(* CODESYS project Rasi_feeds_batching2.project

Project tree, tasks and I/O mapping:
  PLC_AC500_V3 : PM5032-T-ETH, ABB AG, order no. 1SAP123400R0x72, version 3.7.0.0
    application Application
      libraries: ModbusRtu, * (ABB); Util, * (System)
      task Task (cyclic, interval t#10ms, priority 14, watchdog t#20ms x 1) calls batching14
      CheckConfigurationObject
      Diagnosis/
        text list Diag_IO_Bus
        text list Diag_V3_PLC
      global variables GVL
      function block Auto_Batching_V14 [ST]
      function block Semi_Auto_Batching_V14 [ST]
      function block FB_Samyak_Multi [ST]
      function block FB_Samyak_Control [ST]
      function block Auto_Batching_V15 [ST]
      function block Semi_Auto_Batching_V15 [ST]
      program batching14 [FBD]
    OnBoard_IO : 12DI/8DO-T/2DC, ABB AG, version 3.7.0.0
        input  E_Stop_DI : BOOL  // Fast inputs DI0-DI3.Digital input DI0
        input  Main_Cont_FB : BOOL  // Fast inputs DI0-DI3.Digital input DI1
        input  Auto_Mode_FB : BOOL  // Fast inputs DI0-DI3.Digital input DI2
        input  VFD_Run : BOOL  // Fast inputs DI0-DI3.Digital input DI3
        input  Start_PB : BOOL  // Fast inputs DI4-DI7.Digital input DI4
        unmapped channels: Fast inputs DI0-DI3, Fast inputs DI4-DI7, Standard inputs DI8-DI11, Digital inputs - Transistor, Fast outputs DO0-DO3, Fast outputs DO4-DO7, Digital outputs - Transistor
    IO_Bus : I/O-Bus, ABB AG, version 3.7.0.0
    Interfaces : Interfaces, ABB AG, version 3.7.0.0
      TA5142_RS485I : TA5142-RS485I, ABB AG, order no. 1SAP187300R0x02, version 3.7.0.0
        Modbus_RTU_Client : Modbus RTU Client, ABB AG, version 3.7.0.0
      OptionSlot_2
      Ethernet : Ethernet, ABB AG, version 3.7.0.0
        ETH1 : IP Settings, ABB AG, version 3.7.0.0
          NetConfig : NetConfig, ABB AG, version 3.7.0.0
          Modbus_TCP_IP_Server : Modbus TCP/IP Server, ABB AG, version 3.7.0.0
        Protocols : Client Protocols, ABB AG, version 3.7.0.0
    OnBoard_RTC : OnBoard RTC, ABB AG, version 3.7.0.0
  text list GlobalTextList
*)

// PLC_AC500_V3/Application/GVL
{attribute 'qualified_only'}
VAR_GLOBAL
    Recipe_Weights AT %MD100 : ARRAY[1..20] OF REAL;
	Auto_Bin_Material_Mapping AT %MW50: ARRAY[1..6] OF INT;
	Semi_Auto_Bin_Material_Mapping AT %MW60: ARRAY[1..10] OF INT;
	Auto_Coarse_To_Fine_speed AT %MD120: ARRAY[1..6] OF REAL := [1.0,1.0,1.0,1.0,1.0,1.0];
	Semi_Auto_Coarse_To_Fine_speed AT %MD130: ARRAY[1..10] OF REAL := [1.0,1.0,1.0,1.0,1.0,1.0,1.0,1.0,1.0,1.0];
	Auto_Bin_Tolerance AT %MD150: ARRAY[1..6] OF REAL;
	Semi_Auto_Bin_Tolerance AT %MD160: ARRAY[1..10] OF REAL;
	Start_Button AT %MX2.0: BOOL;
	E_Stop_Active AT %MX2.1: BOOL;
	Reset AT %MX2.3: BOOL;
	Next_Cycle_Start AT %MX2.4: BOOL;               // Command pulse/signal to start next batch cycle after hoppers are emptied
	Auto_Active_Mat AT %MW70: INT;
	Auto_Active_Bin AT %MW71: INT;
	Semi_Auto_Active_Mat AT %MW72: INT;
	Semi_Auto_Active_Bin AT %MW73: INT;
	Target_Batch_Cycles AT %MW74: INT := 1;
	Current_Batch_Cycle AT %MW75: INT;
	Completed_Batch_Cycles AT %MW79: INT;
	Error_Code AT %MW76: INT;  // 0=OK 1=DupMat 2=MatRange 3=RecipeLimit 4=ScaleNotEmpty 5=CommunicationFault(Line_Fault) 6=Ex_Weight_Allow_kg_invalid 21=ScaleOverload
	Run AT %MX2.5 : BOOL;
	load_cell_auto AT %MD174 : REAL;
	load_cell_semi_auto AT %MD175 : REAL;
	Auto_Initial_Tolerance AT %MD176 : REAL := 5.0;
	Semi_Auto_Initial_Tolerance AT %MD178 : REAL := 5.0;
	Empty_Weight_Limit AT %MD186 : REAL := 5.0;     // Maximum scale weight limit (kg) to qualify scale as empty before starting next cycle
	Ex_Weight_Allow_kg AT %MD188 : REAL := 0.2;  // Semi-only: oscillation allow (kg) above target; next stage only if actual < Target+Allow
	Auto_Total_Target_Weight AT %MD170 : REAL;
	Semi_Auto_Total_Target_Weight AT %MD171 : REAL;
	Auto_Material_Count AT %MW77: INT;
	Semi_Auto_Material_Count AT %MW78 : INT;
	Auto_Current_Step AT %MW80 : INT;
	Semi_Auto_Current_Step AT %MW81 : INT;
	Auto_Active_Target_Weight AT %MD220 : REAL;
	Semi_Auto_Active_Target_Weight AT %MD224 : REAL;
	Auto_Active_Live_Weight AT %MD172 : REAL;
	Semi_Auto_Active_Live_Weight AT %MD173 : REAL;
	Auto_Excess_Allowed AT %MX2.6: BOOL := 1;
	Semi_Auto_Excess_Allowed AT %MX2.9 : BOOL;
	Auto_Excess_Alarm AT %MX2.7 : BOOL;
	Semi_Auto_Excess_Alarm AT %MX2.8 : BOOL;
	Auto_Inter_Bin_Delay AT %MD190 : TIME;
	Semi_Auto_Inter_Bin_Delay AT %MD194 : TIME;
	Auto_Sequence_Complete AT %MX3.0 : BOOL;
	Semi_Auto_Sequence_Complete AT %MX3.1 : BOOL;
	All_Cycles_Complete AT %MX3.2 : BOOL;           // Master flag: TRUE when all target batch cycles have completed
	Auto_Status_Message : STRING(80);
	Semi_Auto_Status_Message : STRING(80);
	
	(* 8 Process Output and Weight Arrays *)
	Auto_Bin : ARRAY[1..6] OF BOOL;
	auto_bin_cutoff : ARRAY[1..6] OF BOOL;
	auto_bin_motor : ARRAY[1..6] OF BOOL;
	Semi_Auto_Bin : ARRAY[1..10] OF BOOL;
	semi_auto_bin_cutoff : ARRAY[1..10] OF BOOL;
	semi_auto_bin_motor : ARRAY[1..10] OF BOOL;
	Auto_Weights : ARRAY[1..6] OF REAL;
	Semi_Auto_Weights : ARRAY[1..10] OF REAL;
	Waiting_Next_batch_HMI_HIDE AT %MX8.1: BOOL;
END_VAR

// PLC_AC500_V3/Application/batching14
PROGRAM batching14
VAR
	Auto_Ctrl: Auto_Batching_V15;
	Semi_Auto_Ctrl: Semi_Auto_Batching_V15;
	Auto_Complete: BOOL;
	Semi_Auto_Complete: BOOL;
	Auto_Err: INT;
	Auto_Msg: STRING;
	Semi_Auto_Err: INT;
	Semi_Auto_Msg: STRING;
	AutoBatchScale: MODRTUMAST;
	ModEnabler: BLINK;
	SamyakRaw: ARRAY[0..1] OF DINT;
	AutBatchRaw: ARRAY[0..1] OF DINT;
	SemAutoScale: MODRTUMAST;
	SemiAutoScaleRaw: ARRAY[0..1] OF DINT;
	AutoBatchSamyak: REAL;
	FB_Samyak_Multi_1: FB_Samyak_Multi;
	FB_Samyak_Control_1: FB_Samyak_Control;
	Run_PB_1: BOOL;
	Next_Cycle_Start: BOOL;
	TP_1: TP;
	TP_ON: BOOL;
	TP_Out: BOOL;
	TP_Et: TIME;
	arrTare_Cmds: ARRAY[1..4] OF BOOL;
END_VAR

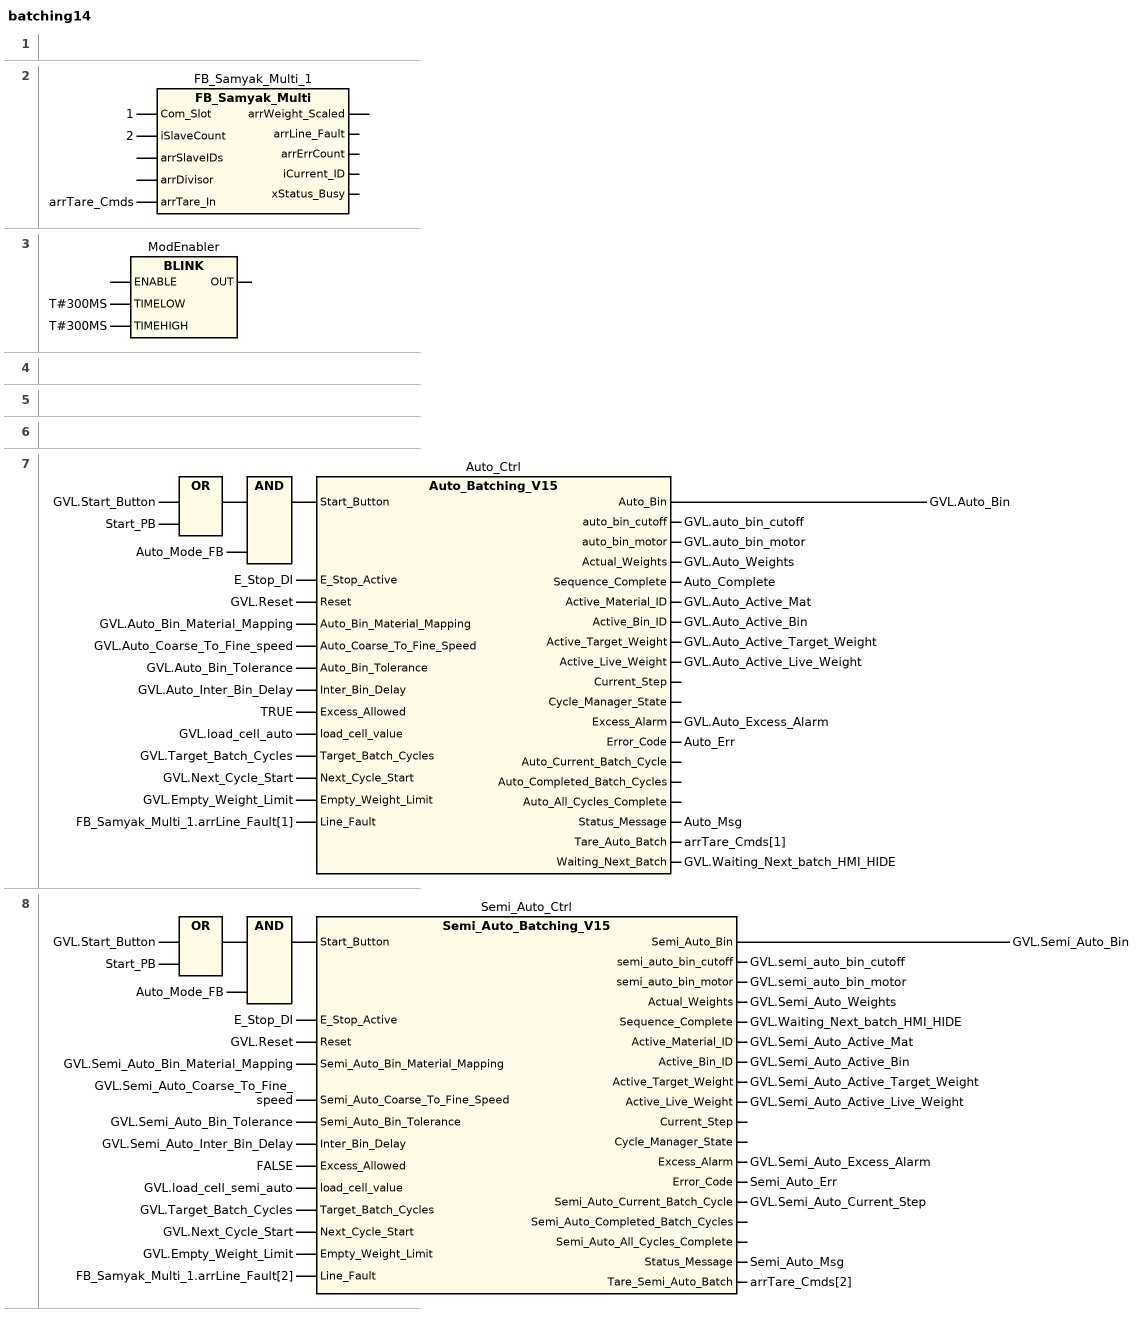
// NETWORK 1

// NETWORK 2
FB_Samyak_Multi_1(Com_Slot := 1, iSlaveCount := 2, arrTare_In := arrTare_Cmds); // FB_Samyak_Multi

// NETWORK 3
ModEnabler(TIMELOW := T#300MS, TIMEHIGH := T#300MS); // BLINK

// NETWORK 4

// NETWORK 5

// NETWORK 6

// NETWORK 7
Auto_Ctrl(
    Start_Button := (GVL.Start_Button OR Start_PB) AND Auto_Mode_FB,
    E_Stop_Active := E_Stop_DI,
    Reset := GVL.Reset,
    Auto_Bin_Material_Mapping := GVL.Auto_Bin_Material_Mapping,
    Auto_Coarse_To_Fine_Speed := GVL.Auto_Coarse_To_Fine_speed,
    Auto_Bin_Tolerance := GVL.Auto_Bin_Tolerance,
    Inter_Bin_Delay := GVL.Auto_Inter_Bin_Delay,
    Excess_Allowed := TRUE,
    load_cell_value := GVL.load_cell_auto,
    Target_Batch_Cycles := GVL.Target_Batch_Cycles,
    Next_Cycle_Start := GVL.Next_Cycle_Start,
    Empty_Weight_Limit := GVL.Empty_Weight_Limit,
    Line_Fault := FB_Samyak_Multi_1.arrLine_Fault[1],
    auto_bin_cutoff => GVL.auto_bin_cutoff,
    auto_bin_motor => GVL.auto_bin_motor,
    Actual_Weights => GVL.Auto_Weights,
    Sequence_Complete => Auto_Complete,
    Active_Material_ID => GVL.Auto_Active_Mat,
    Active_Bin_ID => GVL.Auto_Active_Bin,
    Active_Target_Weight => GVL.Auto_Active_Target_Weight,
    Active_Live_Weight => GVL.Auto_Active_Live_Weight,
    Excess_Alarm => GVL.Auto_Excess_Alarm,
    Error_Code => Auto_Err,
    Status_Message => Auto_Msg,
    Tare_Auto_Batch => arrTare_Cmds[1],
    Waiting_Next_Batch => GVL.Waiting_Next_batch_HMI_HIDE); // Auto_Batching_V15
GVL.Auto_Bin := Auto_Ctrl.Auto_Bin;

// NETWORK 8
Semi_Auto_Ctrl(
    Start_Button := (GVL.Start_Button OR Start_PB) AND Auto_Mode_FB,
    E_Stop_Active := E_Stop_DI,
    Reset := GVL.Reset,
    Semi_Auto_Bin_Material_Mapping := GVL.Semi_Auto_Bin_Material_Mapping,
    Semi_Auto_Coarse_To_Fine_Speed := GVL.Semi_Auto_Coarse_To_Fine_speed,
    Semi_Auto_Bin_Tolerance := GVL.Semi_Auto_Bin_Tolerance,
    Inter_Bin_Delay := GVL.Semi_Auto_Inter_Bin_Delay,
    Excess_Allowed := FALSE,
    load_cell_value := GVL.load_cell_semi_auto,
    Target_Batch_Cycles := GVL.Target_Batch_Cycles,
    Next_Cycle_Start := GVL.Next_Cycle_Start,
    Empty_Weight_Limit := GVL.Empty_Weight_Limit,
    Line_Fault := FB_Samyak_Multi_1.arrLine_Fault[2],
    semi_auto_bin_cutoff => GVL.semi_auto_bin_cutoff,
    semi_auto_bin_motor => GVL.semi_auto_bin_motor,
    Actual_Weights => GVL.Semi_Auto_Weights,
    Sequence_Complete => GVL.Waiting_Next_batch_HMI_HIDE,
    Active_Material_ID => GVL.Semi_Auto_Active_Mat,
    Active_Bin_ID => GVL.Semi_Auto_Active_Bin,
    Active_Target_Weight => GVL.Semi_Auto_Active_Target_Weight,
    Active_Live_Weight => GVL.Semi_Auto_Active_Live_Weight,
    Excess_Alarm => GVL.Semi_Auto_Excess_Alarm,
    Error_Code => Semi_Auto_Err,
    Semi_Auto_Current_Batch_Cycle => GVL.Semi_Auto_Current_Step,
    Status_Message => Semi_Auto_Msg,
    Tare_Semi_Auto_Batch => arrTare_Cmds[2]); // Semi_Auto_Batching_V15
GVL.Semi_Auto_Bin := Semi_Auto_Ctrl.Semi_Auto_Bin;

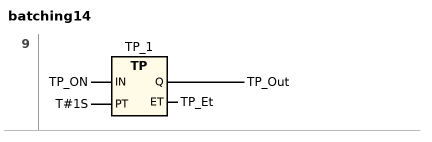
// NETWORK 9
TP_1(IN := TP_ON, PT := T#1S, ET => TP_Et); // TP
TP_Out := TP_1.Q;

END_PROGRAM

// PLC_AC500_V3/Application/FB_Samyak_Multi
//SAMYAK 4016 Multi Slave Unit Customised Block
//Note: This FB_Samyak_Multi name is impotrtant when you create new POU.

FUNCTION_BLOCK FB_Samyak_Multi
VAR_INPUT
    Com_Slot      : BYTE := 1;    (* Port Number *)
    iSlaveCount   : INT := 1;     (* How many slaves active: 1 to 4 *)
    arrSlaveIDs   : ARRAY[1..4] OF BYTE := [1, 2, 3, 4]; (* Unit IDs *)
    arrDivisor    : ARRAY[1..4] OF REAL := [10.0, 10.0, 10.0, 10.0]; (* Scaling per Unit *)
    arrTare_In    : ARRAY[1..4] OF BOOL; (* Individual Tare triggers *)
END_VAR

VAR_OUTPUT
    arrWeight_Scaled : ARRAY[1..4] OF REAL; (* Scaled result per unit *)
    arrLine_Fault    : ARRAY[1..4] OF BOOL; (* Fault status per unit *)
    arrErrCount      : ARRAY[1..4] OF INT;  (* Error count per unit *)
    iCurrent_ID      : BYTE;                (* Current ID being polled *)
    xStatus_Busy     : BOOL;                (* Overall Bus Busy *)
END_VAR

VAR
    (* Internal ModRtuMast Instances *)
    fbRead         : ModRtuMast;
    fbTare         : ModRtuMast;
    
    (* Polling Control *)
    iStep          : INT := 0;
    iIdx           : INT := 1;    (* Current Loop Index *)
    Samyak_Buffer  : ARRAY[0..17] OF WORD;
    wTareCommand   : WORD := 1;
    
    (* Unique Timer/Trigger Instances *)
    rtTareTrig     : R_TRIG;
    rtErrTrig      : R_TRIG;
    tWatchdog      : TON;
    tRecovery      : TON;
END_VAR



(* --- 1. INDIVIDUAL UNIT MONITORING --- *)
iCurrent_ID := arrSlaveIDs[iIdx]; 

(* Watchdog for Bus Hangs *)
tWatchdog(IN := (fbRead.Busy OR fbTare.Busy), PT := T#2000MS);
xStatus_Busy := fbRead.Busy OR fbTare.Busy;

(* Error Tracking for Current Index *)
rtErrTrig(CLK := (fbRead.Error OR fbTare.Error));
IF rtErrTrig.Q THEN
    arrErrCount[iIdx] := arrErrCount[iIdx] + 1;
END_IF

(* Reset on Success *)
IF fbRead.Done OR fbTare.Done THEN
    arrErrCount[iIdx] := 0;
    arrLine_Fault[iIdx] := FALSE;
END_IF

(* Line Fault Activation (10 errors) *)
IF arrErrCount[iIdx] >= 10 THEN
    arrLine_Fault[iIdx] := TRUE;
END_IF

(* Auto-Recovery pulse (5s) *)
tRecovery(IN := arrLine_Fault[iIdx], PT := T#5S);
IF tRecovery.Q THEN
    arrErrCount[iIdx] := 0;
    arrLine_Fault[iIdx] := FALSE;
END_IF

IF tWatchdog.Q THEN iStep := 99; END_IF

(* Check Tare for active slave *)
rtTareTrig(CLK := arrTare_In[iIdx]);

(* --- 2. SEQUENTIAL STATE MACHINE --- *)
CASE iStep OF
    
    0: (* READ CURRENT SLAVE *)
        fbTare(Execute := FALSE);
        fbRead(
            Execute := NOT (fbRead.Done OR fbRead.Error OR fbRead.Busy) 
                       AND NOT rtTareTrig.Q AND NOT arrLine_Fault[iIdx],
            COM     := Com_Slot,
            Serv    := arrSlaveIDs[iIdx],
            FCT     := 3, Addr := 0, Nb := 2, 
            Data    := ADR(Samyak_Buffer[0]), Timeout := 400
        );

        IF fbRead.Done THEN
            (* Scale weight using the array-based divisor for this specific index *)
            arrWeight_Scaled[iIdx] := TO_REAL(TO_DINT(SHL(TO_DWORD(Samyak_Buffer[1]), 16) OR TO_DWORD(Samyak_Buffer[0]))) / arrDivisor[iIdx];
            iStep := 10; (* Switch to next slave *)
        END_IF
        
        IF fbRead.Error THEN iStep := 10; END_IF (* Move on if error *)
        IF rtTareTrig.Q THEN iStep := 1; END_IF  (* Priority: Tare current unit *)

    1: (* PORT RELEASE *)
        fbRead(Execute := FALSE);
        IF NOT fbRead.Busy THEN iStep := 2; END_IF

    2: (* WRITE TARE FOR CURRENT SLAVE *)
        fbTare(
            Execute := TRUE,
            COM := Com_Slot, Serv := arrSlaveIDs[iIdx], 
            FCT := 6, Addr := 16, Nb := 1,
            Data := ADR(wTareCommand), Timeout := 1000
        );

        IF fbTare.Done OR fbTare.Error THEN
            arrTare_In[iIdx] := FALSE; (* Reset manual trigger *)
            iStep := 3;
        END_IF

    3: (* CLEANUP *)
        fbTare(Execute := FALSE);
        IF NOT fbTare.Busy THEN iStep := 10; END_IF

    10: (* INDEX ROTATION *)
        iIdx := iIdx + 1;
        IF iIdx > iSlaveCount THEN
            iIdx := 1; (* Back to first slave *)
        END_IF
        iStep := 0;

    99: (* EMERGENCY RESET *)
        fbRead(Execute := FALSE); fbTare(Execute := FALSE);
        IF NOT (fbRead.Busy OR fbTare.Busy) THEN iStep := 0; END_IF
        
END_CASE

END_FUNCTION_BLOCK

// PLC_AC500_V3/Application/Auto_Batching_V15
FUNCTION_BLOCK Auto_Batching_V15
VAR_INPUT
    Start_Button : BOOL;                            // Command pulse/signal to start or resume the auto batching sequence
    E_Stop_Active : BOOL;                           // Emergency Stop circuit status (NC contact: TRUE = Healthy/Run permitted, FALSE = E-Stop tripped)
    Reset : BOOL;                                   // System reset pulse (clears active steps, outputs, alarms, and error flags)
    Auto_Bin_Material_Mapping : ARRAY[1..6] OF INT; // Array mapping physical Silos 1..6 to Recipe Material IDs (1..20, 0 = Silo skipped)
    Auto_Coarse_To_Fine_Speed : ARRAY[1..6] OF REAL;// Weight offset threshold (kg) before target to transition from Coarse to Fine feeding
    Auto_Bin_Tolerance : ARRAY[1..6] OF REAL;       // Allowable weight tolerance window (±kg) around target weight for each silo
    Inter_Bin_Delay : TIME;                         // Settling delay duration after completing a bin before advancing to the next
    Excess_Allowed : BOOL;                          // Overfill handling policy: TRUE = proceed if target is exceeded, FALSE = raise alarm and halt
    load_cell_value : REAL;                         // Live gross weight input reading from the Auto scale load cell (kg)
    Target_Batch_Cycles : INT;                      // Target number of batch cycle repetitions configured from HMI (defaults to 1)
    Next_Cycle_Start : BOOL;                        // NextBatchStart: after a completed cycle (Target>1), press when this FB scale < Empty_Weight_Limit
    Empty_Weight_Limit : REAL;                      // Tank minimum / empty limit (kg): load_cell must be LT this before Next_Cycle_Start is accepted
    Line_Fault : BOOL;                              // Wire from FB_Samyak_Multi.arrLine_Fault[n] (Auto scale). TRUE = hold process (Over Dump Avoid)
END_VAR
VAR_OUTPUT
    Auto_Bin : ARRAY[1..6] OF BOOL;                 // Coarse feeding valve / gate actuation command outputs for Silos 1..6
    auto_bin_cutoff : ARRAY[1..6] OF BOOL;          // Fine feeding valve / vibrator cutoff actuation command outputs for Silos 1..6
    auto_bin_motor : ARRAY[1..6] OF BOOL;           // Feeder / screw conveyor motor run commands for Silos 1..6
    Actual_Weights : ARRAY[1..6] OF REAL;           // Net material weight (kg) successfully dosed for each silo in the current cycle
    Sequence_Complete : BOOL;                       // Handshake flag: TRUE when all mapped Auto silos have completed dosing and settling
    Active_Material_ID : INT;                       // Recipe Material ID currently being dosed (1..20, 0 when idle/complete)
    Active_Bin_ID : INT;                            // Physical Silo index currently being dosed (1..6, 0 when idle/complete)
    Active_Target_Weight : REAL;                    // Target weight setpoint (kg) of the ingredient currently being dosed
    Active_Live_Weight : REAL;                      // Live net/tared weight (kg) accumulated into the scale for the active silo
    Current_Step : INT;                             // Real-time sequence step:
                                                    //   0  = Idle / Waiting for Start
                                                    //   1..6 = Dosing Silos 1..6 (feeding coarse/fine)
                                                    //   7  = Settling delay in progress
                                                    //   8  = Sequence complete
    Cycle_Manager_State : INT;                      // Master supervisory cycle manager state:
                                                    //   0  = System Idle / Stopped
                                                    //   1  = Running active batch cycle
                                                    //   4  = All target batch cycles completed successfully
                                                    //   5  = Paused between cycles (Cycle Hold active)
    Excess_Alarm : BOOL;                            // Overfill alarm: TRUE when dosed weight exceeds target + tolerance (with Excess_Allowed=FALSE)
    Error_Code : INT;                               // Fault diagnostic code:
                                                    //   0  = No Error / System Healthy
                                                    //   1  = Duplicate Material ID mapped across Auto and Semi-Auto
                                                    //   2  = Material index out of range (must be 1..20)
                                                    //   3  = Recipe weight is less than (Coarse_To_Fine_Speed + Tolerance)
                                                    //   4  = Initial scale tare error (scale not empty before start)
                                                    //   5  = Communication Fault (Line_Fault from FB_Samyak_Multi; scale Modbus/line fault; Over Dump Avoid HOLD)
                                                    //   21 = Scale overload protection triggered (> 500 kg)
    Auto_Current_Batch_Cycle : INT;                     // Active batch cycle number currently processing (1..Target_Batch_Cycles)
    Auto_Completed_Batch_Cycles : INT;                  // Total number of batch cycle loops completed successfully
    Auto_All_Cycles_Complete : BOOL;                    // Master flag: TRUE when all Target_Batch_Cycles have finished
    Status_Message : STRING(80);                    // Real-time human-readable process status and diagnostic text message
    Tare_Auto_Batch : BOOL;                         // One-scan pulse to Samyak arrTare_In[n] at each batch cycle start when scale < Empty_Weight_Limit
    Waiting_Next_Batch : BOOL;                      // TRUE while between cycles waiting for Next_Cycle_Start (Current < Target); FALSE when next cycle runs; never TRUE on last cycle
END_VAR
VAR
    bin_last_weight : REAL;
    actual_bin : REAL;
    target_weight : REAL;
    cutoff_trigger_weight : REAL;
    min_tol_weight : REAL;
    max_tol_weight : REAL;
    Paused_By_EStop : BOOL;
    Effective_Delay : TIME;
    Mat_Idx : INT;
    i : INT;
    j : INT;
    Transition_Timer : TON;
    Completion_Timer : TON;
    Simulation_Mode : BOOL;
    Sim_Rate : REAL;
    Sim_Timer : TON;
    Start_Sim_Weight : REAL;
    Discharge_Active : BOOL;
    
    (* Master Cycle Manager & Supervisory states *)
    Internal_FB_Start : BOOL;
    Duplicate_Found : BOOL;
    Invalid_Material_Range : BOOL;
    Weight_Limit_Error : BOOL;
    eff_empty_limit : REAL;
    Next_Cycle_Last : BOOL;
    Next_Cycle_Rising : BOOL;
    Paused_By_LineFault : BOOL;                     // Latched while Line_Fault is TRUE (outputs forced OFF)
    Tare_Pulse_Req : BOOL;                          // Internal request to emit Tare_Auto_Batch for one scan
END_VAR



(* Auto Batching FB V15: V14 + Line_Fault HOLD (Over Dump Avoid) + Tare_Auto_Batch pulse *)

Effective_Delay := Inter_Bin_Delay;
IF Effective_Delay = T#0S THEN
    Effective_Delay := T#2S;
END_IF;

(* Detect rising edge on Next_Cycle_Start / NextBatchStart (pin OR GVL.%MX2.4) *)
Next_Cycle_Rising := (Next_Cycle_Start OR GVL.Next_Cycle_Start) AND NOT Next_Cycle_Last;
Next_Cycle_Last := (Next_Cycle_Start OR GVL.Next_Cycle_Start);

(* 1. RECIPE TOTALS & SUPERVISORY CONFIGURATION CHECKS *)
Duplicate_Found := FALSE;
Invalid_Material_Range := FALSE;
Weight_Limit_Error := FALSE;

GVL.Auto_Total_Target_Weight := 0.0;
GVL.Auto_Material_Count := 0;
FOR i := 1 TO 6 DO
    IF Auto_Bin_Material_Mapping[i] < 0 OR Auto_Bin_Material_Mapping[i] > 20 THEN
        Invalid_Material_Range := TRUE;
    END_IF;
    IF Auto_Bin_Material_Mapping[i] <> 0 AND Auto_Bin_Material_Mapping[i] <= 20 THEN
        FOR j := 1 TO 10 DO
            IF Auto_Bin_Material_Mapping[i] = GVL.Semi_Auto_Bin_Material_Mapping[j] THEN
                Duplicate_Found := TRUE;
            END_IF;
        END_FOR;
    END_IF;
    IF Auto_Bin_Material_Mapping[i] > 0 AND Auto_Bin_Material_Mapping[i] <= 20 THEN
        IF GVL.Recipe_Weights[Auto_Bin_Material_Mapping[i]] > 0.0 THEN
            GVL.Auto_Total_Target_Weight := GVL.Auto_Total_Target_Weight + GVL.Recipe_Weights[Auto_Bin_Material_Mapping[i]];
            GVL.Auto_Material_Count := GVL.Auto_Material_Count + 1;
            IF GVL.Recipe_Weights[Auto_Bin_Material_Mapping[i]] < (Auto_Coarse_To_Fine_Speed[i] + Auto_Bin_Tolerance[i]) THEN
                Weight_Limit_Error := TRUE;
            END_IF;
        END_IF;
    END_IF;
END_FOR;

IF Duplicate_Found THEN
    GVL.Error_Code := 1;
    Error_Code := 1;
    Status_Message := 'Error 1: Duplicate Material ID mapped in Auto and Semi-Auto!';
ELSIF Invalid_Material_Range THEN
    GVL.Error_Code := 2;
    Error_Code := 2;
    Status_Message := 'Error 2: Material Index configuration out of range (1..20)!';
ELSIF Weight_Limit_Error THEN
    GVL.Error_Code := 3;
    Error_Code := 3;
    Status_Message := 'Error 3: Recipe weight is less than Coarse_To_Fine_Speed + Tolerance!';
ELSE
    IF GVL.Error_Code <= 3 THEN
        GVL.Error_Code := 0;
        Error_Code := 0;
    END_IF;
END_IF;

(* 2. HARD RESET INTERLOCK *)
IF Reset OR GVL.Reset THEN
    FOR i := 1 TO 6 DO
        Auto_Bin[i] := FALSE;
        auto_bin_cutoff[i] := FALSE;
        auto_bin_motor[i] := FALSE;
        Actual_Weights[i] := 0.0;
        GVL.Auto_Bin[i] := FALSE;
        GVL.auto_bin_cutoff[i] := FALSE;
        GVL.auto_bin_motor[i] := FALSE;
        GVL.Auto_Weights[i] := 0.0;
    END_FOR;
    
    (* Reset Recipe & Active Target Setpoints *)
    FOR i := 1 TO 20 DO
        GVL.Recipe_Weights[i] := 0.0;
    END_FOR;
    GVL.Auto_Total_Target_Weight := 0.0;
    GVL.Semi_Auto_Total_Target_Weight := 0.0;
    GVL.Auto_Material_Count := 0;
    GVL.Semi_Auto_Material_Count := 0;
    
    Sequence_Complete := FALSE;
    GVL.Auto_Sequence_Complete := FALSE;
    GVL.Semi_Auto_Sequence_Complete := FALSE;
    Active_Material_ID := 0;
    Active_Bin_ID := 0;
    Active_Target_Weight := 0.0;
    Active_Live_Weight := 0.0;
    GVL.Auto_Active_Target_Weight := 0.0;
    GVL.Auto_Active_Live_Weight := 0.0;
    Excess_Alarm := FALSE;
    Error_Code := 0;
    GVL.Error_Code := 0;
    GVL.Current_Batch_Cycle := 0;
    GVL.Completed_Batch_Cycles := 0;
    GVL.All_Cycles_Complete := FALSE;
    Auto_Completed_Batch_Cycles := 0;
    Auto_Current_Batch_Cycle := 0;
    Auto_All_Cycles_Complete := FALSE;
    GVL.Target_Batch_Cycles := 0;
    GVL.Start_Button := FALSE;
    GVL.Run := FALSE;
    GVL.Next_Cycle_Start := FALSE;
    Next_Cycle_Last := FALSE;
    Next_Cycle_Rising := FALSE;
    GVL.Auto_Active_Mat := 0;
    GVL.Auto_Active_Bin := 0;
    GVL.Auto_Excess_Alarm := FALSE;
    Current_Step := 0;
    Cycle_Manager_State := 0;
    Internal_FB_Start := FALSE;
    Paused_By_LineFault := FALSE;
    Tare_Pulse_Req := FALSE;
    Tare_Auto_Batch := FALSE;
    Waiting_Next_Batch := FALSE;
    bin_last_weight := 0.0;
    Start_Sim_Weight := 0.0;
    Transition_Timer(IN := FALSE);
    Completion_Timer(IN := FALSE);
    Sim_Timer(IN := FALSE);
    Status_Message := 'Auto [Reset]: System Reset Complete - System Idle';
    RETURN;
END_IF;

(* 3. E-STOP PAUSE / HOLD LOGIC (NC Contact: FALSE = Pressed/Tripped, TRUE = Healthy) *)
IF NOT E_Stop_Active OR NOT GVL.E_Stop_Active THEN
    Paused_By_EStop := TRUE;
END_IF;

IF Paused_By_EStop THEN
    FOR i := 1 TO 6 DO
        Auto_Bin[i] := FALSE;
        auto_bin_cutoff[i] := FALSE;
        auto_bin_motor[i] := FALSE;
    END_FOR;
    IF NOT E_Stop_Active OR NOT GVL.E_Stop_Active THEN
        Status_Message := CONCAT('Auto [PAUSED]: E-Stop Active at Step ', INT_TO_STRING(Current_Step));
    ELSE
        Status_Message := CONCAT('Auto [HOLD]: E-Stop Cleared. Press Start to Resume Step ', INT_TO_STRING(Current_Step));
        IF Start_Button OR GVL.Start_Button THEN
            Paused_By_EStop := FALSE;
        END_IF;
    END_IF;
    Sim_Timer(IN := FALSE);
    Transition_Timer(IN := FALSE);
    Completion_Timer(IN := FALSE);
    RETURN;
END_IF;

(* 3b. LINE FAULT HOLD — Over Dump Avoid (wire Line_Fault from FB_Samyak_Multi.arrLine_Fault[n]) *)
(* While scale comms/line is faulted, freeze sequence and force feed outputs OFF. Auto-resume when fault clears. *)
Tare_Auto_Batch := FALSE;
IF Line_Fault THEN
    Paused_By_LineFault := TRUE;
END_IF;

IF Paused_By_LineFault THEN
    FOR i := 1 TO 6 DO
        Auto_Bin[i] := FALSE;
        auto_bin_cutoff[i] := FALSE;
        auto_bin_motor[i] := FALSE;
    END_FOR;
    Tare_Auto_Batch := FALSE;
    IF Line_Fault THEN
        Error_Code := 5; (* Communication Fault *)
        GVL.Error_Code := 5;
        Status_Message := CONCAT('Auto [HOLD]: Error 5 Communication Fault (Line_Fault) at Step ', INT_TO_STRING(Current_Step));
    ELSE
        Paused_By_LineFault := FALSE;
        IF Error_Code = 5 THEN
            Error_Code := 0;
        END_IF;
        IF GVL.Error_Code = 5 THEN
            GVL.Error_Code := 0;
        END_IF;
        Status_Message := CONCAT('Auto [RESUME]: Communication Fault cleared - continuing Step ', INT_TO_STRING(Current_Step));
    END_IF;
    Sim_Timer(IN := FALSE);
    Transition_Timer(IN := FALSE);
    Completion_Timer(IN := FALSE);
    RETURN;
END_IF;

(* 4. MASTER CYCLE MANAGER STATE MACHINE *)
CASE Cycle_Manager_State OF
    0: (* IDLE *)
        Internal_FB_Start := FALSE;
        GVL.Run := FALSE;
        GVL.Next_Cycle_Start := FALSE;
        GVL.Auto_Sequence_Complete := FALSE;
        
        IF GVL.Error_Code = 0 AND NOT (Start_Button OR GVL.Start_Button) THEN
            Status_Message := 'Auto [State 0 - Idle]: Ready - Waiting for Start Button';
        END_IF;
        
        IF Start_Button OR GVL.Start_Button THEN
            (* Use Target_Batch_Cycles from input, or fallback to GVL, or default to 1 *)
            IF Target_Batch_Cycles > 0 THEN
                GVL.Target_Batch_Cycles := Target_Batch_Cycles;
            ELSIF GVL.Target_Batch_Cycles <= 0 THEN
                GVL.Target_Batch_Cycles := 1;
            END_IF;
            
            IF NOT E_Stop_Active OR NOT GVL.E_Stop_Active THEN
                GVL.Run := FALSE;
                Status_Message := 'Auto [State 0]: Cannot Start - Emergency Stop Contact Open!';
            ELSIF (GVL.Auto_Initial_Tolerance > 0.0 AND (GVL.load_cell_auto > GVL.Auto_Initial_Tolerance OR GVL.load_cell_auto < (-GVL.Auto_Initial_Tolerance))) OR 
                  (GVL.Semi_Auto_Initial_Tolerance > 0.0 AND (GVL.load_cell_semi_auto > GVL.Semi_Auto_Initial_Tolerance OR GVL.load_cell_semi_auto < (-GVL.Semi_Auto_Initial_Tolerance))) THEN
                GVL.Run := FALSE;
                GVL.Error_Code := 4;
                Error_Code := 4;
                Status_Message := 'Auto [State 0]: Error 4 - Scale not zeroed (exceeds Initial Tolerance)!';
            ELSE
                GVL.Error_Code := 0;
                Error_Code := 0;
                GVL.Current_Batch_Cycle := 1;
                GVL.Completed_Batch_Cycles := 0;
                GVL.All_Cycles_Complete := FALSE;
                Auto_Completed_Batch_Cycles := 0;
                Auto_Current_Batch_Cycle := 1;
                Auto_All_Cycles_Complete := FALSE;
                GVL.Run := TRUE;
                Internal_FB_Start := TRUE;
                Cycle_Manager_State := 1;
                Current_Step := 0;
                Tare_Pulse_Req := TRUE; (* Pulse Tare_Auto_Batch if scale empty *)
            END_IF;
        END_IF;
        
    1: (* RUNNING CYCLE *)
        Internal_FB_Start := TRUE;
        GVL.Run := TRUE;
        
        (* Interlock: While process is actively running, Next_Cycle_Start MUST be FALSE *)
        GVL.Next_Cycle_Start := FALSE;
        
        (* Both Auto and Semi-Auto must complete to finish the cycle *)
        IF Sequence_Complete AND GVL.Semi_Auto_Sequence_Complete THEN
            GVL.Completed_Batch_Cycles := GVL.Current_Batch_Cycle;
            Auto_Completed_Batch_Cycles := GVL.Current_Batch_Cycle;
            IF GVL.Current_Batch_Cycle < GVL.Target_Batch_Cycles AND GVL.Error_Code = 0 THEN
                Internal_FB_Start := FALSE;
                Cycle_Manager_State := 5; (* Go to pause/hold to wait for scale empty & Next_Cycle_Start *)
            ELSE
                Cycle_Manager_State := 4; (* All target cycles completed *)
            END_IF;
        END_IF;
        
    5: (* PAUSED BETWEEN CYCLES — Next_Cycle_Start / NextBatchStart *)
        (* Purpose: Target_Batch_Cycles > 1 AND at least one cycle completed (Completed >= 1)
           AND more cycles remain (Completed < Target). Operator empties tank (load_cell LT
           Empty_Weight_Limit), then presses Next_Cycle_Start. Same rule as Semi FB. *)
        Internal_FB_Start := FALSE;
        GVL.Run := TRUE;
        
        (* Tank minimum weight / empty threshold (default 5.0 kg if unset) *)
        eff_empty_limit := Empty_Weight_Limit;
        IF eff_empty_limit <= 0.0 THEN
            eff_empty_limit := GVL.Empty_Weight_Limit;
        END_IF;
        IF eff_empty_limit <= 0.0 THEN
            eff_empty_limit := 5.0;
        END_IF;
        
        Status_Message := CONCAT('Auto [State 5]: Cycle ', CONCAT(INT_TO_STRING(GVL.Current_Batch_Cycle), ' Done. Empty scale < limit then Next_Cycle_Start.'));
        
        (* Accept ONLY on rising edge of Next_Cycle_Start (pin OR GVL) *)
        IF Next_Cycle_Rising THEN
            IF (GVL.Target_Batch_Cycles > 1) AND (GVL.Completed_Batch_Cycles >= 1) AND (GVL.Completed_Batch_Cycles < GVL.Target_Batch_Cycles) THEN
                (* This FB scale must be LT tank minimum; also require Semi scale empty so both sides agree *)
                IF (load_cell_value < eff_empty_limit) AND (GVL.load_cell_semi_auto < eff_empty_limit) THEN
                    (* Do NOT clear GVL.Next_Cycle_Start here — Semi runs later same scan and must see the pulse.
                       State 1 interlock clears it on the next scan. *)
                    GVL.Start_Button := TRUE; (* Keep Start_Button TRUE until all cycles are complete! *)
                    GVL.Error_Code := 0;
                    Error_Code := 0;
                    GVL.Current_Batch_Cycle := GVL.Current_Batch_Cycle + 1;
                    Auto_Current_Batch_Cycle := GVL.Current_Batch_Cycle;
                    Sequence_Complete := FALSE;
                    GVL.Auto_Sequence_Complete := FALSE;
                    GVL.Semi_Auto_Sequence_Complete := FALSE;
                    Current_Step := 0;
                    Internal_FB_Start := TRUE;
                    Cycle_Manager_State := 1;
                    Tare_Pulse_Req := TRUE; (* Pulse Tare_Auto_Batch if scale empty before next cycle *)
                    FOR i := 1 TO 6 DO
                        Actual_Weights[i] := 0.0;
                        Auto_Bin[i] := FALSE;
                        auto_bin_cutoff[i] := FALSE;
                        auto_bin_motor[i] := FALSE;
                    END_FOR;
                ELSE
                    (* Scale not empty: reject, clear command so operator can press again after emptying *)
                    GVL.Next_Cycle_Start := FALSE;
                    Next_Cycle_Last := FALSE;
                    Status_Message := CONCAT('Auto [State 5]: Scale >= limit (', CONCAT(REAL_TO_STRING(eff_empty_limit), ' kg)! Empty then Next_Cycle_Start again.'));
                END_IF;
            ELSE
                GVL.Next_Cycle_Start := FALSE;
                Next_Cycle_Last := FALSE;
                Status_Message := 'Auto [State 5]: Next_Cycle_Start ignored (need Target>1 and Completed>=1 and Completed<Target)';
            END_IF;
        END_IF;
        
    4: (* ALL CYCLES COMPLETE *)
        Internal_FB_Start := FALSE;
        GVL.Run := FALSE;
        GVL.Start_Button := FALSE;
        Auto_All_Cycles_Complete := TRUE;
        GVL.All_Cycles_Complete := TRUE;
        Sequence_Complete := TRUE;
        GVL.Auto_Sequence_Complete := TRUE;
        GVL.Semi_Auto_Sequence_Complete := TRUE;
        Status_Message := CONCAT('Auto [State 4 - Finished]: All ', CONCAT(INT_TO_STRING(GVL.Target_Batch_Cycles), ' Batch Cycles Completed Successfully'));
        IF Start_Button OR GVL.Start_Button THEN
            (* Reset flags for new batch start *)
            Current_Step := 0;
            Auto_All_Cycles_Complete := FALSE;
            GVL.All_Cycles_Complete := FALSE;
            Sequence_Complete := FALSE;
            GVL.Auto_Sequence_Complete := FALSE;
            GVL.Semi_Auto_Sequence_Complete := FALSE;
            Cycle_Manager_State := 0;
        END_IF;
END_CASE;

(* Waiting_Next_Batch: TRUE only in between-cycle hold while Current < Target
   Example Target=3: after cycle 1 done (Current=1) → TRUE; next cycle starts → FALSE;
   after cycle 2 done (Current=2) → TRUE; when Current=3 (last) → never TRUE. *)
Waiting_Next_Batch := (Cycle_Manager_State = 5)
    AND (GVL.Target_Batch_Cycles > 1)
    AND (GVL.Current_Batch_Cycle < GVL.Target_Batch_Cycles);

(* 4b. TARE PULSE — one scan TRUE to FB_Samyak_Multi.arrTare_In[n] when starting a cycle from ~0 kg *)
IF Tare_Pulse_Req THEN
    eff_empty_limit := Empty_Weight_Limit;
    IF eff_empty_limit <= 0.0 THEN
        eff_empty_limit := GVL.Empty_Weight_Limit;
    END_IF;
    IF eff_empty_limit <= 0.0 THEN
        eff_empty_limit := 5.0;
    END_IF;
    IF load_cell_value < eff_empty_limit THEN
        Tare_Auto_Batch := TRUE;
        Status_Message := 'Auto [Tare]: Scale empty - Tare_Auto_Batch pulse issued';
    ELSE
        Tare_Auto_Batch := FALSE;
        Status_Message := CONCAT('Auto [Tare skipped]: Scale not empty (>= ', CONCAT(REAL_TO_STRING(eff_empty_limit), ' kg)'));
    END_IF;
    Tare_Pulse_Req := FALSE;
END_IF;

(* 5. AUTO SILOS 1..6 POURING SEQUENCE WITH DETAILED STATUS *)
IF Current_Step = 0 AND Internal_FB_Start THEN
    Current_Step := 1;
    bin_last_weight := load_cell_value;
    Sequence_Complete := FALSE;
    GVL.Auto_Sequence_Complete := FALSE;
    Excess_Alarm := FALSE;
    Error_Code := 0;
    FOR i := 1 TO 6 DO
        Actual_Weights[i] := 0.0;
        Auto_Bin[i] := FALSE;
        auto_bin_cutoff[i] := FALSE;
        auto_bin_motor[i] := FALSE;
    END_FOR;
END_IF;

CASE Current_Step OF
    0:
        Active_Material_ID := 0;
        Active_Bin_ID := 0;
        Excess_Alarm := FALSE;
        Sequence_Complete := FALSE;
        FOR i := 1 TO 6 DO
            Auto_Bin[i] := FALSE;
            auto_bin_cutoff[i] := FALSE;
            auto_bin_motor[i] := FALSE;
        END_FOR;
        Active_Target_Weight := GVL.Auto_Active_Target_Weight;
        Active_Live_Weight := 0.0;
        
    1..6:
        (* Skip any bin where Material Mapping is 0, > 20, or Recipe Weight is 0 *)
        WHILE Current_Step >= 1 AND Current_Step <= 6 DO
            Mat_Idx := Auto_Bin_Material_Mapping[Current_Step];
            IF Mat_Idx = 0 OR Mat_Idx > 20 OR GVL.Recipe_Weights[Mat_Idx] <= 0.0 THEN
                Auto_Bin[Current_Step] := FALSE;
                auto_bin_cutoff[Current_Step] := FALSE;
                auto_bin_motor[Current_Step] := FALSE;
                Actual_Weights[Current_Step] := 0.0;
                IF Current_Step = 6 THEN
                    Current_Step := 7;
                    EXIT;
                ELSE
                    Current_Step := Current_Step + 1;
                END_IF;
            ELSE
                EXIT; (* Valid active recipe silo found *)
            END_IF;
        END_WHILE;
        
        IF Current_Step = 7 THEN
            Active_Material_ID := 0;
            Active_Bin_ID := 0;
            Active_Target_Weight := 0.0;
            Active_Live_Weight := 0.0;
            GVL.Auto_Active_Target_Weight := 0.0;
            GVL.Auto_Active_Live_Weight := 0.0;
            Status_Message := 'Auto [Step 7]: Settling Delay in progress...';
            Completion_Timer(IN := TRUE, PT := Effective_Delay);
            IF Completion_Timer.Q THEN
                Completion_Timer(IN := FALSE);
                Current_Step := 8;
            END_IF;
        ELSE
            Mat_Idx := Auto_Bin_Material_Mapping[Current_Step];
            target_weight := GVL.Recipe_Weights[Mat_Idx];
            
            Active_Target_Weight := target_weight;
            GVL.Auto_Active_Target_Weight := target_weight;
            
            cutoff_trigger_weight := target_weight - Auto_Coarse_To_Fine_Speed[Current_Step];
            min_tol_weight := target_weight - Auto_Bin_Tolerance[Current_Step];
            max_tol_weight := target_weight + Auto_Bin_Tolerance[Current_Step];
            
            actual_bin := load_cell_value - bin_last_weight;
            IF actual_bin < 0.0 THEN
                actual_bin := 0.0;
            END_IF;
            Actual_Weights[Current_Step] := actual_bin;
            Active_Live_Weight := actual_bin;
            GVL.Auto_Active_Live_Weight := actual_bin;
            Active_Material_ID := Mat_Idx;
            Active_Bin_ID := Current_Step;
            
            IF load_cell_value > 500.0 THEN
                Error_Code := 21;
                GVL.Error_Code := 21;
                Status_Message := CONCAT('Auto [Step ', CONCAT(INT_TO_STRING(Current_Step), ']: STUCK - Error 21: Scale Overloaded (> 500 kg)!'));
                Sequence_Complete := TRUE;
                GVL.Auto_Sequence_Complete := TRUE;
                Paused_By_EStop := TRUE;
            END_IF;
            
            IF actual_bin < cutoff_trigger_weight THEN
                Auto_Bin[Current_Step] := TRUE;
                auto_bin_cutoff[Current_Step] := FALSE;
                auto_bin_motor[Current_Step] := TRUE;
                Excess_Alarm := FALSE;
                Status_Message := CONCAT('Auto [Step ', CONCAT(INT_TO_STRING(Current_Step), ']: Coarse Feeding'));
            ELSIF actual_bin < min_tol_weight THEN
                Auto_Bin[Current_Step] := FALSE;
                auto_bin_cutoff[Current_Step] := TRUE;
                auto_bin_motor[Current_Step] := TRUE;
                Excess_Alarm := FALSE;
                Status_Message := CONCAT('Auto [Step ', CONCAT(INT_TO_STRING(Current_Step), ']: Fine Feeding'));
            ELSIF actual_bin > max_tol_weight THEN
                Auto_Bin[Current_Step] := FALSE;
                auto_bin_cutoff[Current_Step] := FALSE;
                auto_bin_motor[Current_Step] := FALSE;
                IF Excess_Allowed THEN
                    Excess_Alarm := FALSE;
                    Status_Message := CONCAT('Auto [Step ', CONCAT(INT_TO_STRING(Current_Step), ']: Excess Allowed - Advancing'));
                    bin_last_weight := load_cell_value;
                    Active_Target_Weight := 0.0;
                    Active_Live_Weight := 0.0;
                    GVL.Auto_Active_Target_Weight := 0.0;
                    GVL.Auto_Active_Live_Weight := 0.0;
                    IF Current_Step = 6 THEN
                        Current_Step := 7;
                    ELSE
                        Current_Step := Current_Step + 1;
                    END_IF;
                ELSE
                    Excess_Alarm := TRUE;
                    Status_Message := CONCAT('Auto [Step ', CONCAT(INT_TO_STRING(Current_Step), ']: STUCK - Excess Weight! Reduce weight or enable Excess Allowed.'));
                END_IF;
            ELSE
                Auto_Bin[Current_Step] := FALSE;
                auto_bin_cutoff[Current_Step] := FALSE;
                auto_bin_motor[Current_Step] := FALSE;
                Excess_Alarm := FALSE;
                bin_last_weight := load_cell_value;
                Active_Target_Weight := 0.0;
                Active_Live_Weight := 0.0;
                GVL.Auto_Active_Target_Weight := 0.0;
                GVL.Auto_Active_Live_Weight := 0.0;
                Status_Message := CONCAT('Auto [Step ', CONCAT(INT_TO_STRING(Current_Step), ']: Target Reached - Advancing'));
                IF Current_Step = 6 THEN
                    Current_Step := 7;
                ELSE
                    Current_Step := Current_Step + 1;
                END_IF;
            END_IF;
        END_IF;

    7:
        Active_Material_ID := 0;
        Active_Bin_ID := 0;
        Excess_Alarm := FALSE;
        Status_Message := 'Auto [Step 7]: Settling Delay in progress...';
        Completion_Timer(IN := TRUE, PT := Effective_Delay);
        IF Completion_Timer.Q THEN
            Completion_Timer(IN := FALSE);
            Current_Step := 8;
        END_IF;
        
    8:
        Active_Material_ID := 0;
        Active_Bin_ID := 0;
        Excess_Alarm := FALSE;
        Sequence_Complete := TRUE;
        GVL.Auto_Sequence_Complete := TRUE;
        IF NOT GVL.Semi_Auto_Sequence_Complete THEN
            Status_Message := 'Auto [Step 8]: Auto Finished. Waiting for Semi-Auto to complete...';
        ELSE
            Status_Message := 'Auto [Step 8]: Cycle Sequences Complete';
        END_IF;
END_CASE;

(* Synchronize physical output arrays to GVL *)
FOR i := 1 TO 6 DO
    GVL.Auto_Bin[i] := Auto_Bin[i];
    GVL.auto_bin_cutoff[i] := auto_bin_cutoff[i];
    GVL.auto_bin_motor[i] := auto_bin_motor[i];
END_FOR;

(* Synchronize live cycle progress to outputs *)
Auto_Current_Batch_Cycle := GVL.Current_Batch_Cycle;
Auto_Completed_Batch_Cycles := GVL.Completed_Batch_Cycles;
Auto_All_Cycles_Complete := GVL.All_Cycles_Complete;

END_FUNCTION_BLOCK

// PLC_AC500_V3/Application/Semi_Auto_Batching_V15
FUNCTION_BLOCK Semi_Auto_Batching_V15
VAR_INPUT
    Start_Button : BOOL;                                 // Command pulse/signal to start or resume the semi-auto batching sequence
    E_Stop_Active : BOOL;                                // Emergency Stop circuit status (NC contact: TRUE = Healthy/Run permitted, FALSE = E-Stop tripped)
    Reset : BOOL;                                        // System reset pulse (clears active steps, outputs, alarms, and error flags)
    Semi_Auto_Bin_Material_Mapping : ARRAY[1..10] OF INT;// Array mapping physical Silos 1..10 to Recipe Material IDs (1..20, 0 = Silo skipped)
    Semi_Auto_Coarse_To_Fine_Speed : ARRAY[1..10] OF REAL;// Weight offset threshold (kg) before target to transition from Coarse to Fine feeding
    Semi_Auto_Bin_Tolerance : ARRAY[1..10] OF REAL;      // Allowable weight tolerance window (±kg) around target weight for each silo
    Inter_Bin_Delay : TIME;                              // Settling delay duration after completing a bin before advancing to the next
    Excess_Allowed : BOOL;                               // Overfill handling policy: TRUE = proceed if target is exceeded, FALSE = raise alarm and halt
    load_cell_value : REAL;                              // Live gross weight input reading from the Semi-Auto scale load cell (kg)
    Target_Batch_Cycles : INT;                           // Target number of batch cycle repetitions configured from HMI (defaults to 1)
    Next_Cycle_Start : BOOL;                             // NextBatchStart: after a completed cycle (Target>1), press when this FB scale < Empty_Weight_Limit
    Empty_Weight_Limit : REAL;                           // Tank minimum / empty limit (kg): load_cell must be LT this before Next_Cycle_Start is accepted
    Line_Fault : BOOL;                                   // Wire from FB_Samyak_Multi.arrLine_Fault[n] (Semi scale). TRUE = hold process (Over Dump Avoid)
END_VAR
VAR_OUTPUT
    Semi_Auto_Bin : ARRAY[1..10] OF BOOL;                // Coarse feeding valve / gate actuation command outputs for Silos 1..10
    semi_auto_bin_cutoff : ARRAY[1..10] OF BOOL;         // Fine feeding valve / vibrator cutoff actuation command outputs for Silos 1..10
    semi_auto_bin_motor : ARRAY[1..10] OF BOOL;          // Feeder / screw conveyor motor run commands for Silos 1..10
    Actual_Weights : ARRAY[1..10] OF REAL;               // Net material weight (kg) successfully dosed for each silo in the current cycle
    Sequence_Complete : BOOL;                            // Handshake flag: TRUE when all mapped Semi-Auto silos have completed dosing and settling
    Active_Material_ID : INT;                            // Recipe Material ID currently being dosed (1..20, 0 when idle/complete)
    Active_Bin_ID : INT;                                 // Physical Silo index currently being dosed (1..10, 0 when idle/complete)
    Active_Target_Weight : REAL;                         // Target weight setpoint (kg) of the ingredient currently being dosed
    Active_Live_Weight : REAL;                           // Live net/tared weight (kg) accumulated into the scale for the active silo
    Current_Step : INT;                                  // Real-time sequence step:
                                                         //   0   = Idle / Waiting for Start
                                                         //   1..10 = Dosing Silos 1..10 (feeding coarse/fine)
                                                         //   31  = Settling delay in progress
                                                         //   32  = Sequence complete
    Cycle_Manager_State : INT;                           // Master supervisory cycle manager state:
                                                         //   0   = System Idle / Stopped
                                                         //   1   = Running active batch cycle
                                                         //   4   = All target batch cycles completed successfully
                                                         //   5   = Paused between cycles (Cycle Hold active)
    Excess_Alarm : BOOL;                                 // Overfill alarm: TRUE when weight > Target+Tolerance and Excess_Allowed=FALSE (clears when weight back in band)
    Error_Code : INT;                                    // Fault diagnostic code:
                                                         //   0   = No Error / System Healthy
                                                         //   1   = Duplicate Material ID mapped across Auto and Semi-Auto
                                                         //   2   = Material index out of range (must be 1..20)
                                                         //   3   = Recipe weight is less than (Coarse_To_Fine_Speed + Tolerance)
                                                         //   4   = Initial scale tare error (scale not empty before start)
                                                         //   5   = Communication Fault (Line_Fault from FB_Samyak_Multi; scale Modbus/line fault; Over Dump Avoid HOLD)
                                                         //   21  = Scale overload protection triggered (> 500 kg)
    Semi_Auto_Current_Batch_Cycle : INT;                 // Active batch cycle number currently processing (1..Target_Batch_Cycles)
    Semi_Auto_Completed_Batch_Cycles : INT;              // Total number of batch cycle loops completed successfully
    Semi_Auto_All_Cycles_Complete : BOOL;                // Master flag: TRUE when all Target_Batch_Cycles have finished
    Status_Message : STRING(80);                         // Real-time human-readable process status and diagnostic text message
    Tare_Semi_Auto_Batch : BOOL;                         // One-scan pulse to Samyak arrTare_In[n] at each batch cycle start when scale < Empty_Weight_Limit
END_VAR
VAR
    bin_last_weight : REAL;
    actual_bin : REAL;
    target_weight : REAL;
    cutoff_trigger_weight : REAL;
    min_tol_weight : REAL;
    max_tol_weight : REAL;
    Paused_By_EStop : BOOL;
    Effective_Delay : TIME;
    Mat_Idx : INT;
    i : INT;
    Last_Batch_Cycle : INT;
    Transition_Timer : TON;
    Completion_Timer : TON;
    Simulation_Mode : BOOL;
    Sim_Rate : REAL;
    Sim_Timer : TON;
    Start_Sim_Weight : REAL;
    Discharge_Active : BOOL;
    Run_Last : BOOL;
    Run_Rising : BOOL;
    Next_Cycle_Last : BOOL;                              // Edge memory for Next_Cycle_Start (same as Auto FB)
    Next_Cycle_Rising : BOOL;                            // Rising edge of Next_Cycle_Start OR GVL.Next_Cycle_Start
    Between_Cycle_Hold : BOOL;                           // TRUE while waiting for empty scale + Next_Cycle_Start (state 5)
    Paused_By_LineFault : BOOL;                          // Latched while Line_Fault is TRUE (outputs forced OFF)
    Tare_Pulse_Req : BOOL;                               // Internal request to emit Tare_Semi_Auto_Batch for one scan
    eff_empty_limit : REAL;
END_VAR



(* Semi-Auto Batching FB V15: Line_Fault HOLD + Tare pulse + Next_Cycle_Start; Excess = same V14 tolerance logic *)

Effective_Delay := Inter_Bin_Delay;
IF Effective_Delay = T#0S THEN
    Effective_Delay := T#2S;
END_IF;

(* Detect rising edge on Next_Cycle_Start trigger — same as Auto FB *)
Next_Cycle_Rising := (Next_Cycle_Start OR GVL.Next_Cycle_Start) AND NOT Next_Cycle_Last;
Next_Cycle_Last := (Next_Cycle_Start OR GVL.Next_Cycle_Start);

(* Track Master Cycle State *)
IF Target_Batch_Cycles > 0 THEN
    GVL.Target_Batch_Cycles := Target_Batch_Cycles;
END_IF;

(* Master Cycle State & Start Synchronization *)
Run_Rising := GVL.Run AND NOT Run_Last;
Run_Last := GVL.Run;

IF GVL.Run THEN
    IF Sequence_Complete AND GVL.Auto_Sequence_Complete THEN
        IF GVL.Current_Batch_Cycle >= GVL.Target_Batch_Cycles AND GVL.Target_Batch_Cycles > 0 THEN
            Cycle_Manager_State := 4;
            Between_Cycle_Hold := FALSE;
        ELSE
            (* More cycles remain — enter / stay in between-cycle hold (state 5) *)
            Cycle_Manager_State := 5;
            Between_Cycle_Hold := TRUE;
        END_IF;
    ELSIF Between_Cycle_Hold THEN
        (* Stay in state 5 until Next_Cycle_Start accepted (empty scale + rising edge) *)
        Cycle_Manager_State := 5;
    ELSE
        Cycle_Manager_State := 1;
    END_IF;
ELSE
    Cycle_Manager_State := 0;
    Current_Step := 0;
    Last_Batch_Cycle := 0;
    Sequence_Complete := FALSE;
    GVL.Semi_Auto_Sequence_Complete := FALSE;
    Between_Cycle_Hold := FALSE;
END_IF;

(* On fresh batch start (rising edge of Run), ensure clean start from Step 0 *)
IF Run_Rising THEN
    Current_Step := 0;
    Last_Batch_Cycle := 0;
    Sequence_Complete := FALSE;
    GVL.Semi_Auto_Sequence_Complete := FALSE;
    Tare_Pulse_Req := TRUE; (* Pulse Tare_Semi_Auto_Batch if scale empty at cycle start *)
END_IF;

(* 1. SEMI-AUTO RECIPE TOTALS & ACTIVE SILO COUNT *)
GVL.Semi_Auto_Total_Target_Weight := 0.0;
GVL.Semi_Auto_Material_Count := 0;
FOR i := 1 TO 10 DO
    IF Semi_Auto_Bin_Material_Mapping[i] > 0 AND Semi_Auto_Bin_Material_Mapping[i] <= 20 THEN
        IF GVL.Recipe_Weights[Semi_Auto_Bin_Material_Mapping[i]] > 0.0 THEN
            GVL.Semi_Auto_Total_Target_Weight := GVL.Semi_Auto_Total_Target_Weight + GVL.Recipe_Weights[Semi_Auto_Bin_Material_Mapping[i]];
            GVL.Semi_Auto_Material_Count := GVL.Semi_Auto_Material_Count + 1;
        END_IF;
    END_IF;
END_FOR;

(* 2. HARD RESET INTERLOCK *)
IF Reset OR GVL.Reset THEN
    FOR i := 1 TO 10 DO
        Semi_Auto_Bin[i] := FALSE;
        semi_auto_bin_cutoff[i] := FALSE;
        semi_auto_bin_motor[i] := FALSE;
        Actual_Weights[i] := 0.0;
        GVL.Semi_Auto_Bin[i] := FALSE;
        GVL.semi_auto_bin_cutoff[i] := FALSE;
        GVL.semi_auto_bin_motor[i] := FALSE;
        GVL.Semi_Auto_Weights[i] := 0.0;
    END_FOR;
    Sequence_Complete := FALSE;
    GVL.Semi_Auto_Sequence_Complete := FALSE;
    Active_Material_ID := 0;
    Active_Bin_ID := 0;
    Active_Target_Weight := 0.0;
    Active_Live_Weight := 0.0;
    GVL.Semi_Auto_Active_Target_Weight := 0.0;
    GVL.Semi_Auto_Active_Live_Weight := 0.0;
    GVL.Semi_Auto_Active_Mat := 0;
    GVL.Semi_Auto_Active_Bin := 0;
    GVL.Semi_Auto_Excess_Alarm := FALSE;
    Excess_Alarm := FALSE;
    Error_Code := 0;
    Paused_By_EStop := FALSE;
    Current_Step := 0;
    Last_Batch_Cycle := 0;
    Cycle_Manager_State := 0;
    Semi_Auto_Current_Batch_Cycle := 0;
    Semi_Auto_Completed_Batch_Cycles := 0;
    Semi_Auto_All_Cycles_Complete := FALSE;
    bin_last_weight := 0.0;
    Start_Sim_Weight := 0.0;
    Run_Last := FALSE;
    Run_Rising := FALSE;
    Next_Cycle_Last := FALSE;
    Next_Cycle_Rising := FALSE;
    Between_Cycle_Hold := FALSE;
    Paused_By_LineFault := FALSE;
    Tare_Pulse_Req := FALSE;
    Tare_Semi_Auto_Batch := FALSE;
    Transition_Timer(IN := FALSE);
    Completion_Timer(IN := FALSE);
    Sim_Timer(IN := FALSE);
    Status_Message := 'Semi-Auto [Reset]: System Reset Complete - System Idle';
    
    (* Clean Auto-Clearing: Reset has been processed by both blocks *)
    GVL.Reset := FALSE;
    RETURN;
END_IF;

(* 3. E-STOP PAUSE / HOLD LOGIC (NC Contact: FALSE = Pressed/Tripped, TRUE = Healthy) *)
IF NOT E_Stop_Active OR NOT GVL.E_Stop_Active THEN
    Paused_By_EStop := TRUE;
END_IF;

IF Paused_By_EStop THEN
    FOR i := 1 TO 10 DO
        Semi_Auto_Bin[i] := FALSE;
        semi_auto_bin_cutoff[i] := FALSE;
        semi_auto_bin_motor[i] := FALSE;
    END_FOR;
    IF NOT E_Stop_Active OR NOT GVL.E_Stop_Active THEN
        Status_Message := CONCAT('Semi-Auto [PAUSED]: E-Stop Active at Step ', INT_TO_STRING(Current_Step));
    ELSE
        Status_Message := CONCAT('Semi-Auto [HOLD]: E-Stop Cleared. Press Start to Resume Step ', INT_TO_STRING(Current_Step));
        IF Start_Button OR GVL.Start_Button THEN
            Paused_By_EStop := FALSE;
        END_IF;
    END_IF;
    Sim_Timer(IN := FALSE);
    Transition_Timer(IN := FALSE);
    Completion_Timer(IN := FALSE);
    RETURN;
END_IF;

(* 3b. LINE FAULT HOLD — Over Dump Avoid (wire Line_Fault from FB_Samyak_Multi.arrLine_Fault[n]) *)
Tare_Semi_Auto_Batch := FALSE;
IF Line_Fault THEN
    Paused_By_LineFault := TRUE;
END_IF;

IF Paused_By_LineFault THEN
    FOR i := 1 TO 10 DO
        Semi_Auto_Bin[i] := FALSE;
        semi_auto_bin_cutoff[i] := FALSE;
        semi_auto_bin_motor[i] := FALSE;
    END_FOR;
    Tare_Semi_Auto_Batch := FALSE;
    IF Line_Fault THEN
        Error_Code := 5; (* Communication Fault *)
        GVL.Error_Code := 5;
        Status_Message := CONCAT('Semi-Auto [HOLD]: Error 5 Communication Fault (Line_Fault) at Step ', INT_TO_STRING(Current_Step));
    ELSE
        Paused_By_LineFault := FALSE;
        IF Error_Code = 5 THEN
            Error_Code := 0;
        END_IF;
        IF GVL.Error_Code = 5 THEN
            GVL.Error_Code := 0;
        END_IF;
        Status_Message := CONCAT('Semi-Auto [RESUME]: Communication Fault cleared - continuing Step ', INT_TO_STRING(Current_Step));
    END_IF;
    Sim_Timer(IN := FALSE);
    Transition_Timer(IN := FALSE);
    Completion_Timer(IN := FALSE);
    RETURN;
END_IF;

(* 3c. TARE PULSE — one scan TRUE to FB_Samyak_Multi.arrTare_In[n] when starting a cycle from ~0 kg *)
IF Tare_Pulse_Req THEN
    eff_empty_limit := Empty_Weight_Limit;
    IF eff_empty_limit <= 0.0 THEN
        eff_empty_limit := GVL.Empty_Weight_Limit;
    END_IF;
    IF eff_empty_limit <= 0.0 THEN
        eff_empty_limit := 5.0;
    END_IF;
    IF load_cell_value < eff_empty_limit THEN
        Tare_Semi_Auto_Batch := TRUE;
        Status_Message := 'Semi-Auto [Tare]: Scale empty - Tare_Semi_Auto_Batch pulse issued';
    ELSE
        Tare_Semi_Auto_Batch := FALSE;
        Status_Message := CONCAT('Semi-Auto [Tare skipped]: Scale not empty (>= ', CONCAT(REAL_TO_STRING(eff_empty_limit), ' kg)'));
    END_IF;
    Tare_Pulse_Req := FALSE;
END_IF;

(* 4. BETWEEN-CYCLE HOLD — Next_Cycle_Start / NextBatchStart (same rule as Auto FB) *)
(* Purpose: Target_Batch_Cycles > 1 AND Completed_Batch_Cycles >= 1 AND Completed < Target.
   Operator empties THIS FB scale (load_cell LT Empty_Weight_Limit), then presses Next_Cycle_Start.
   Auto FB advances GVL.Current_Batch_Cycle; Semi releases hold and restarts dosing. *)
IF Cycle_Manager_State = 5 OR Between_Cycle_Hold THEN
    Cycle_Manager_State := 5;
    eff_empty_limit := Empty_Weight_Limit;
    IF eff_empty_limit <= 0.0 THEN
        eff_empty_limit := GVL.Empty_Weight_Limit;
    END_IF;
    IF eff_empty_limit <= 0.0 THEN
        eff_empty_limit := 5.0;
    END_IF;

    Status_Message := 'Semi-Auto [State 5]: Empty scale < limit then press Next_Cycle_Start';

    IF Next_Cycle_Rising THEN
        IF (GVL.Target_Batch_Cycles > 1) AND (GVL.Completed_Batch_Cycles >= 1) AND (GVL.Completed_Batch_Cycles < GVL.Target_Batch_Cycles) THEN
            IF load_cell_value < eff_empty_limit THEN
                (* Accept: release hold. Do not clear GVL.Next_Cycle_Start (Auto may still need pulse same scan). *)
                Between_Cycle_Hold := FALSE;
                Sequence_Complete := FALSE;
                GVL.Semi_Auto_Sequence_Complete := FALSE;
                Current_Step := 0;
                Last_Batch_Cycle := GVL.Current_Batch_Cycle;
                Tare_Pulse_Req := TRUE;
                Excess_Alarm := FALSE;
                Error_Code := 0;
                FOR i := 1 TO 10 DO
                    Actual_Weights[i] := 0.0;
                    Semi_Auto_Bin[i] := FALSE;
                    semi_auto_bin_cutoff[i] := FALSE;
                    semi_auto_bin_motor[i] := FALSE;
                END_FOR;
                Cycle_Manager_State := 1;
                Status_Message := 'Semi-Auto [State 5]: Next_Cycle_Start accepted — starting next cycle';
            ELSE
                (* Reject: clear command so operator can press again after emptying *)
                GVL.Next_Cycle_Start := FALSE;
                Next_Cycle_Last := FALSE;
                Status_Message := CONCAT('Semi-Auto [State 5]: Scale >= limit (', CONCAT(REAL_TO_STRING(eff_empty_limit), ' kg)! Empty then Next_Cycle_Start again.'));
            END_IF;
        ELSE
            GVL.Next_Cycle_Start := FALSE;
            Next_Cycle_Last := FALSE;
            Status_Message := 'Semi-Auto [State 5]: Next_Cycle_Start ignored (need Target>1 and Completed>=1 and Completed<Target)';
        END_IF;
    END_IF;
END_IF;

(* 5. SEQUENCE START (FOR CYCLE 1 AND REPEAT CYCLES) *)
IF GVL.Run AND Cycle_Manager_State <> 5 AND NOT Between_Cycle_Hold THEN
    IF Current_Step = 0 THEN
        Last_Batch_Cycle := GVL.Current_Batch_Cycle;
        Current_Step := 1;
        bin_last_weight := load_cell_value;
        Sequence_Complete := FALSE;
        GVL.Semi_Auto_Sequence_Complete := FALSE;
        Excess_Alarm := FALSE;
        Error_Code := 0;
        FOR i := 1 TO 10 DO
            Actual_Weights[i] := 0.0;
            Semi_Auto_Bin[i] := FALSE;
            semi_auto_bin_cutoff[i] := FALSE;
            semi_auto_bin_motor[i] := FALSE;
        END_FOR;
    ELSIF Current_Step = 32 AND GVL.Current_Batch_Cycle <> Last_Batch_Cycle THEN
        (* Advance to next cycle loop (Cycle 2, 3, etc.) — cycle number already bumped by Auto *)
        Last_Batch_Cycle := GVL.Current_Batch_Cycle;
        Tare_Pulse_Req := TRUE; (* next-cycle tare if empty — emit next scan before dosing *)
        Current_Step := 0; (* return to Step 0 so tare pulse runs before Step 1 *)
        bin_last_weight := load_cell_value;
        Sequence_Complete := FALSE;
        GVL.Semi_Auto_Sequence_Complete := FALSE;
        Excess_Alarm := FALSE;
        Error_Code := 0;
        FOR i := 1 TO 10 DO
            Actual_Weights[i] := 0.0;
            Semi_Auto_Bin[i] := FALSE;
            semi_auto_bin_cutoff[i] := FALSE;
            semi_auto_bin_motor[i] := FALSE;
        END_FOR;
    END_IF;
END_IF;

CASE Current_Step OF
    0:
        Active_Material_ID := 0;
        Active_Bin_ID := 0;
        Excess_Alarm := FALSE;
        Sequence_Complete := FALSE;
        FOR i := 1 TO 10 DO
            Semi_Auto_Bin[i] := FALSE;
            semi_auto_bin_cutoff[i] := FALSE;
            semi_auto_bin_motor[i] := FALSE;
        END_FOR;
        Active_Target_Weight := GVL.Semi_Auto_Active_Target_Weight;
        Active_Live_Weight := 0.0;
        IF Error_Code = 0 AND Cycle_Manager_State <> 5 THEN 
            Status_Message := 'Semi-Auto [Step 0 - Idle]: Ready - Waiting for Run Signal'; 
        END_IF;
        
    1..10:
        (* Skip any bin where Material Mapping is 0, > 20, or Recipe Weight is 0 *)
        WHILE Current_Step >= 1 AND Current_Step <= 10 DO
            Mat_Idx := Semi_Auto_Bin_Material_Mapping[Current_Step];
            IF Mat_Idx = 0 OR Mat_Idx > 20 OR GVL.Recipe_Weights[Mat_Idx] <= 0.0 THEN
                Semi_Auto_Bin[Current_Step] := FALSE;
                semi_auto_bin_cutoff[Current_Step] := FALSE;
                semi_auto_bin_motor[Current_Step] := FALSE;
                Actual_Weights[Current_Step] := 0.0;
                IF Current_Step = 10 THEN
                    Current_Step := 31;
                    EXIT;
                ELSE
                    Current_Step := Current_Step + 1;
                END_IF;
            ELSE
                EXIT; (* Valid active recipe silo found *)
            END_IF;
        END_WHILE;
        
        IF Current_Step = 31 THEN
            Active_Material_ID := 0;
            Active_Bin_ID := 0;
            Active_Target_Weight := 0.0;
            Active_Live_Weight := 0.0;
            GVL.Semi_Auto_Active_Target_Weight := 0.0;
            GVL.Semi_Auto_Active_Live_Weight := 0.0;
            Status_Message := 'Semi-Auto [Step 31]: Settling Delay in progress...';
            Completion_Timer(IN := TRUE, PT := Effective_Delay);
            IF Completion_Timer.Q THEN
                Completion_Timer(IN := FALSE);
                Current_Step := 32;
            END_IF;
        ELSE
            Mat_Idx := Semi_Auto_Bin_Material_Mapping[Current_Step];
            target_weight := GVL.Recipe_Weights[Mat_Idx];
            
            Active_Target_Weight := target_weight;
            GVL.Semi_Auto_Active_Target_Weight := target_weight;
            
            cutoff_trigger_weight := target_weight - Semi_Auto_Coarse_To_Fine_Speed[Current_Step];
            min_tol_weight := target_weight - Semi_Auto_Bin_Tolerance[Current_Step]; (* e.g. 10.0 - 0.2 = 9.8 *)
            max_tol_weight := target_weight + Semi_Auto_Bin_Tolerance[Current_Step]; (* e.g. 10.0 + 0.2 = 10.2 *)
            
            actual_bin := load_cell_value - bin_last_weight;
            IF actual_bin < 0.0 THEN
                actual_bin := 0.0;
            END_IF;
            Actual_Weights[Current_Step] := actual_bin; (* keeps live value, e.g. 15 kg if overfill with Excess_Allowed *)
            Active_Live_Weight := actual_bin;
            GVL.Semi_Auto_Active_Live_Weight := actual_bin;
            Active_Material_ID := Mat_Idx;
            Active_Bin_ID := Current_Step;
            
            IF load_cell_value > 500.0 THEN
                Error_Code := 21;
                GVL.Error_Code := 21;
                Status_Message := CONCAT('Semi-Auto [Step ', CONCAT(INT_TO_STRING(Current_Step), ']: STUCK - Error 21: Scale Overloaded (> 500 kg)!'));
                Sequence_Complete := TRUE;
                GVL.Semi_Auto_Sequence_Complete := TRUE;
                Paused_By_EStop := TRUE;
            END_IF;
            
            IF actual_bin < cutoff_trigger_weight THEN
                Semi_Auto_Bin[Current_Step] := TRUE;
                semi_auto_bin_cutoff[Current_Step] := FALSE;
                semi_auto_bin_motor[Current_Step] := TRUE;
                Excess_Alarm := FALSE;
                Status_Message := CONCAT('Semi-Auto [Step ', CONCAT(INT_TO_STRING(Current_Step), ']: Coarse Feeding'));
            ELSIF actual_bin < min_tol_weight THEN
                (* e.g. 9.6 < 9.8 — still fine feeding, Excess_Alarm FALSE *)
                Semi_Auto_Bin[Current_Step] := FALSE;
                semi_auto_bin_cutoff[Current_Step] := TRUE;
                semi_auto_bin_motor[Current_Step] := TRUE;
                Excess_Alarm := FALSE;
                Status_Message := CONCAT('Semi-Auto [Step ', CONCAT(INT_TO_STRING(Current_Step), ']: Fine Feeding'));
            ELSIF actual_bin > max_tol_weight THEN
                (* e.g. GT 10.2 — stop feeders *)
                Semi_Auto_Bin[Current_Step] := FALSE;
                semi_auto_bin_cutoff[Current_Step] := FALSE;
                semi_auto_bin_motor[Current_Step] := FALSE;
                IF Excess_Allowed THEN
                    (* Overfill OK: advance next material; Actual_Weights already shows true weight (e.g. 15 kg) *)
                    Excess_Alarm := FALSE;
                    Status_Message := CONCAT('Semi-Auto [Step ', CONCAT(INT_TO_STRING(Current_Step), ']: Excess Allowed - Advancing'));
                    bin_last_weight := load_cell_value;
                    Active_Target_Weight := 0.0;
                    Active_Live_Weight := 0.0;
                    GVL.Semi_Auto_Active_Target_Weight := 0.0;
                    GVL.Semi_Auto_Active_Live_Weight := 0.0;
                    IF Current_Step = 10 THEN
                        Current_Step := 31;
                    ELSE
                        Current_Step := Current_Step + 1;
                    END_IF;
                ELSE
                    (* Excess_Allowed=FALSE: Excess_Alarm TRUE until weight drops back into tolerance band, then advance *)
                    Excess_Alarm := TRUE;
                    Status_Message := CONCAT('Semi-Auto [Step ', CONCAT(INT_TO_STRING(Current_Step), ']: STUCK - Excess Weight! Reduce weight or enable Excess Allowed.'));
                END_IF;
            ELSE
                (* In band [min_tol .. max_tol], e.g. 9.8..10.2 — advance next material / settle *)
                Semi_Auto_Bin[Current_Step] := FALSE;
                semi_auto_bin_cutoff[Current_Step] := FALSE;
                semi_auto_bin_motor[Current_Step] := FALSE;
                Excess_Alarm := FALSE;
                bin_last_weight := load_cell_value;
                Active_Target_Weight := 0.0;
                Active_Live_Weight := 0.0;
                GVL.Semi_Auto_Active_Target_Weight := 0.0;
                GVL.Semi_Auto_Active_Live_Weight := 0.0;
                Status_Message := CONCAT('Semi-Auto [Step ', CONCAT(INT_TO_STRING(Current_Step), ']: Target Reached - Advancing'));
                IF Current_Step = 10 THEN
                    Current_Step := 31;
                ELSE
                    Current_Step := Current_Step + 1;
                END_IF;
            END_IF;
        END_IF;

    31:
        Active_Material_ID := 0;
        Active_Bin_ID := 0;
        Excess_Alarm := FALSE;
        Status_Message := 'Semi-Auto [Step 31]: Settling Delay in progress...';
        Completion_Timer(IN := TRUE, PT := Effective_Delay);
        IF Completion_Timer.Q THEN
            Completion_Timer(IN := FALSE);
            Current_Step := 32;
        END_IF;
        
    32:
        Active_Material_ID := 0;
        Active_Bin_ID := 0;
        Excess_Alarm := FALSE;
        Sequence_Complete := TRUE;
        GVL.Semi_Auto_Sequence_Complete := TRUE;
        IF NOT GVL.Auto_Sequence_Complete THEN
            Status_Message := 'Semi-Auto [Step 32]: Semi-Auto Finished. Waiting for Auto to complete...';
        ELSE
            Status_Message := 'Semi-Auto [Step 32]: Cycle Sequences Complete';
        END_IF;
END_CASE;

(* Synchronize physical output arrays to GVL *)
FOR i := 1 TO 10 DO
    GVL.Semi_Auto_Bin[i] := Semi_Auto_Bin[i];
    GVL.semi_auto_bin_cutoff[i] := semi_auto_bin_cutoff[i];
    GVL.semi_auto_bin_motor[i] := semi_auto_bin_motor[i];
END_FOR;

(* Synchronize live cycle progress to outputs *)
Semi_Auto_Current_Batch_Cycle := GVL.Current_Batch_Cycle;
Semi_Auto_Completed_Batch_Cycles := GVL.Completed_Batch_Cycles;
Semi_Auto_All_Cycles_Complete := GVL.All_Cycles_Complete;

END_FUNCTION_BLOCK

// PLC_AC500_V3/Application/FB_Samyak_Control
FUNCTION_BLOCK FB_Samyak_Control
VAR_INPUT
    Com_Slot      : BYTE := 1;     (* PLC COM port *)
    Slave_Dev_ID  : BYTE := 1;     (* Samyak slave ID *)
    iDivisor      : REAL := 10.0;  (* Scale factor: Weight_Scaled = Raw / iDivisor *)
    xTare_In      : BOOL;           (* Logic tare pulse *)
    xManual_Tare  : BOOL;           (* HMI/manual tare pulse *)
END_VAR

VAR_OUTPUT
    xStatus_Done   : BOOL;
    xStatus_Busy   : BOOL;
    xStatus_Error  : BOOL;
    iTotalErrCount : INT := 0;
    xLine_Fault    : BOOL;
    Weight_Raw     : DINT;
    Weight_Scaled  : REAL;
    wError_Code    : WORD; (* Check PLC & SAMYAK BaudRate, DevId, Parity; also check PLC serial port LED blink status and RS485 connection if error repeats *)
END_VAR

VAR
    fbRead         : ModRtuMast;
    fbTare         : ModRtuMast;
    iStep          : INT := 0;
    Samyak_Buffer  : ARRAY[0..17] OF WORD;
    wTareCommand   : WORD := 1;

    rtTareTrig     : R_TRIG;
    rtErrTrig      : R_TRIG;
    tStuckWatchdog : TON;
    tRecoveryTimer : TON;

    xTareReq       : BOOL := FALSE; (* Internal tare request latch *)
END_VAR


(* --- 1) Error Tracking + Auto Recovery --- *)
tStuckWatchdog(IN := (fbRead.Busy OR fbTare.Busy), PT := T#2000MS);

rtErrTrig(CLK := (fbRead.Error OR fbTare.Error));
IF rtErrTrig.Q THEN
    iTotalErrCount := iTotalErrCount + 1;
END_IF

IF fbRead.Done OR fbTare.Done THEN
    iTotalErrCount := 0;
    xLine_Fault := FALSE;
END_IF

IF iTotalErrCount >= 10 THEN
    xLine_Fault := TRUE;
END_IF

tRecoveryTimer(IN := xLine_Fault, PT := T#5S);
IF tRecoveryTimer.Q THEN
    iTotalErrCount := 0;
    xLine_Fault := FALSE;
END_IF

IF tStuckWatchdog.Q THEN
    iStep := 99;
END_IF

(* Capture tare request from either input pulse *)
rtTareTrig(CLK := xTare_In OR xManual_Tare);
IF rtTareTrig.Q THEN
    xTareReq := TRUE;
END_IF

(* --- 2) Modbus State Machine --- *)
CASE iStep OF

    0:  (* Continuous Read *)
        fbTare(Execute := FALSE);

        fbRead(
            Execute := NOT (fbRead.Done OR fbRead.Error OR fbRead.Busy)
                       AND NOT xTareReq
                       AND NOT xLine_Fault,
            COM     := Com_Slot,
            Serv    := Slave_Dev_ID,
            FCT     := 3,
            Addr    := 0,
            Nb      := 2,
            Data    := ADR(Samyak_Buffer[0]),
            Timeout := 400,
            Done    => xStatus_Done,
            Busy    => xStatus_Busy,
            Error   => xStatus_Error,
            ErrorID => wError_Code
        );

        IF xStatus_Done THEN
            Weight_Raw := TO_DINT(SHL(TO_DWORD(Samyak_Buffer[1]), 16) OR TO_DWORD(Samyak_Buffer[0]));
            Weight_Scaled := TO_REAL(Weight_Raw) / iDivisor;
        END_IF

        IF xTareReq THEN
            iStep := 1;
        END_IF

    1:  (* Port Release *)
        fbRead(Execute := FALSE);
        IF NOT fbRead.Busy THEN
            iStep := 2;
        END_IF

    2:  (* Execute Tare *)
        fbTare(
            Execute := TRUE,
            COM     := Com_Slot,
            Serv    := Slave_Dev_ID,
            FCT     := 6,
            Addr    := 16,
            Nb      := 1,
            Data    := ADR(wTareCommand),
            Timeout := 1000,
            Done    => xStatus_Done,
            Busy    => xStatus_Busy,
            Error   => xStatus_Error,
            ErrorID => wError_Code
        );

        IF fbTare.Done OR fbTare.Error THEN
            xTareReq := FALSE;
            iStep := 3;
        END_IF

    3:  (* Return to Read *)
        fbTare(Execute := FALSE);
        IF NOT fbTare.Busy THEN
            iStep := 0;
        END_IF

    99: (* Emergency Recovery *)
        fbRead(Execute := FALSE);
        fbTare(Execute := FALSE);

        IF NOT (fbRead.Busy OR fbTare.Busy) THEN
            iTotalErrCount := 0;
            iStep := 0;
        END_IF

END_CASE

END_FUNCTION_BLOCK

// PLC_AC500_V3/Application/Auto_Batching_V14
FUNCTION_BLOCK Auto_Batching_V14
VAR_INPUT
    Start_Button : BOOL;                            // Command pulse/signal to start or resume the auto batching sequence
    E_Stop_Active : BOOL;                           // Emergency Stop circuit status (NC contact: TRUE = Healthy/Run permitted, FALSE = E-Stop tripped)
    Reset : BOOL;                                   // System reset pulse (clears active steps, outputs, alarms, and error flags)
    Auto_Bin_Material_Mapping : ARRAY[1..6] OF INT; // Array mapping physical Silos 1..6 to Recipe Material IDs (1..20, 0 = Silo skipped)
    Auto_Coarse_To_Fine_Speed : ARRAY[1..6] OF REAL;// Weight offset threshold (kg) before target to transition from Coarse to Fine feeding
    Auto_Bin_Tolerance : ARRAY[1..6] OF REAL;       // Allowable weight tolerance window (±kg) around target weight for each silo
    Inter_Bin_Delay : TIME;                         // Settling delay duration after completing a bin before advancing to the next
    Excess_Allowed : BOOL;                          // Overfill handling policy: TRUE = proceed if target is exceeded, FALSE = raise alarm and halt
    load_cell_value : REAL;                         // Live gross weight input reading from the Auto scale load cell (kg)
    Target_Batch_Cycles : INT;                      // Target number of batch cycle repetitions configured from HMI (defaults to 1)
    Next_Cycle_Start : BOOL;                        // Command pulse/signal to start next batch cycle after hoppers are emptied
    Empty_Weight_Limit : REAL;                      // Maximum scale weight limit (kg) for scales to qualify as empty before starting next cycle
END_VAR
VAR_OUTPUT
    Auto_Bin : ARRAY[1..6] OF BOOL;                 // Coarse feeding valve / gate actuation command outputs for Silos 1..6
    auto_bin_cutoff : ARRAY[1..6] OF BOOL;          // Fine feeding valve / vibrator cutoff actuation command outputs for Silos 1..6
    auto_bin_motor : ARRAY[1..6] OF BOOL;           // Feeder / screw conveyor motor run commands for Silos 1..6
    Actual_Weights : ARRAY[1..6] OF REAL;           // Net material weight (kg) successfully dosed for each silo in the current cycle
    Sequence_Complete : BOOL;                       // Handshake flag: TRUE when all mapped Auto silos have completed dosing and settling
    Active_Material_ID : INT;                       // Recipe Material ID currently being dosed (1..20, 0 when idle/complete)
    Active_Bin_ID : INT;                            // Physical Silo index currently being dosed (1..6, 0 when idle/complete)
    Active_Target_Weight : REAL;                    // Target weight setpoint (kg) of the ingredient currently being dosed
    Active_Live_Weight : REAL;                      // Live net/tared weight (kg) accumulated into the scale for the active silo
    Current_Step : INT;                             // Real-time sequence step:
                                                    //   0  = Idle / Waiting for Start
                                                    //   1..6 = Dosing Silos 1..6 (feeding coarse/fine)
                                                    //   7  = Settling delay in progress
                                                    //   8  = Sequence complete
    Cycle_Manager_State : INT;                      // Master supervisory cycle manager state:
                                                    //   0  = System Idle / Stopped
                                                    //   1  = Running active batch cycle
                                                    //   4  = All target batch cycles completed successfully
                                                    //   5  = Paused between cycles (Cycle Hold active)
    Excess_Alarm : BOOL;                            // Overfill alarm: TRUE when dosed weight exceeds target + tolerance (with Excess_Allowed=FALSE)
    Error_Code : INT;                               // Fault diagnostic code:
                                                    //   0  = No Error / System Healthy
                                                    //   1  = Duplicate Material ID mapped across Auto and Semi-Auto
                                                    //   2  = Material index out of range (must be 1..20)
                                                    //   3  = Recipe weight is less than (Coarse_To_Fine_Speed + Tolerance)
                                                    //   4  = Initial scale tare error (scale not empty before start)
                                                    //   21 = Scale overload protection triggered (> 500 kg)
    Auto_Current_Batch_Cycle : INT;                     // Active batch cycle number currently processing (1..Target_Batch_Cycles)
    Auto_Completed_Batch_Cycles : INT;                  // Total number of batch cycle loops completed successfully
    Auto_All_Cycles_Complete : BOOL;                    // Master flag: TRUE when all Target_Batch_Cycles have finished
    Status_Message : STRING(80);                    // Real-time human-readable process status and diagnostic text message
END_VAR
VAR
    bin_last_weight : REAL;
    actual_bin : REAL;
    target_weight : REAL;
    cutoff_trigger_weight : REAL;
    min_tol_weight : REAL;
    max_tol_weight : REAL;
    Paused_By_EStop : BOOL;
    Effective_Delay : TIME;
    Mat_Idx : INT;
    i : INT;
    j : INT;
    Transition_Timer : TON;
    Completion_Timer : TON;
    Simulation_Mode : BOOL;
    Sim_Rate : REAL;
    Sim_Timer : TON;
    Start_Sim_Weight : REAL;
    Discharge_Active : BOOL;
    
    (* Master Cycle Manager & Supervisory states *)
    Internal_FB_Start : BOOL;
    Duplicate_Found : BOOL;
    Invalid_Material_Range : BOOL;
    Weight_Limit_Error : BOOL;
    eff_empty_limit : REAL;
    Next_Cycle_Last : BOOL;
    Next_Cycle_Rising : BOOL;
END_VAR


(* Auto Batching FB V14 with Full Diagnostics, Step Tracking, and Precise Status Reporting *)

Effective_Delay := Inter_Bin_Delay;
IF Effective_Delay = T#0S THEN
    Effective_Delay := T#2S;
END_IF;

(* Detect rising edge on Next_Cycle_Start trigger *)
Next_Cycle_Rising := (Next_Cycle_Start OR GVL.Next_Cycle_Start) AND NOT Next_Cycle_Last;
Next_Cycle_Last := (Next_Cycle_Start OR GVL.Next_Cycle_Start);

(* 1. RECIPE TOTALS & SUPERVISORY CONFIGURATION CHECKS *)
Duplicate_Found := FALSE;
Invalid_Material_Range := FALSE;
Weight_Limit_Error := FALSE;

GVL.Auto_Total_Target_Weight := 0.0;
GVL.Auto_Material_Count := 0;
FOR i := 1 TO 6 DO
    IF Auto_Bin_Material_Mapping[i] < 0 OR Auto_Bin_Material_Mapping[i] > 20 THEN
        Invalid_Material_Range := TRUE;
    END_IF;
    IF Auto_Bin_Material_Mapping[i] <> 0 AND Auto_Bin_Material_Mapping[i] <= 20 THEN
        FOR j := 1 TO 10 DO
            IF Auto_Bin_Material_Mapping[i] = GVL.Semi_Auto_Bin_Material_Mapping[j] THEN
                Duplicate_Found := TRUE;
            END_IF;
        END_FOR;
    END_IF;
    IF Auto_Bin_Material_Mapping[i] > 0 AND Auto_Bin_Material_Mapping[i] <= 20 THEN
        IF GVL.Recipe_Weights[Auto_Bin_Material_Mapping[i]] > 0.0 THEN
            GVL.Auto_Total_Target_Weight := GVL.Auto_Total_Target_Weight + GVL.Recipe_Weights[Auto_Bin_Material_Mapping[i]];
            GVL.Auto_Material_Count := GVL.Auto_Material_Count + 1;
            IF GVL.Recipe_Weights[Auto_Bin_Material_Mapping[i]] < (Auto_Coarse_To_Fine_Speed[i] + Auto_Bin_Tolerance[i]) THEN
                Weight_Limit_Error := TRUE;
            END_IF;
        END_IF;
    END_IF;
END_FOR;

IF Duplicate_Found THEN
    GVL.Error_Code := 1;
    Error_Code := 1;
    Status_Message := 'Error 1: Duplicate Material ID mapped in Auto and Semi-Auto!';
ELSIF Invalid_Material_Range THEN
    GVL.Error_Code := 2;
    Error_Code := 2;
    Status_Message := 'Error 2: Material Index configuration out of range (1..20)!';
ELSIF Weight_Limit_Error THEN
    GVL.Error_Code := 3;
    Error_Code := 3;
    Status_Message := 'Error 3: Recipe weight is less than Coarse_To_Fine_Speed + Tolerance!';
ELSE
    IF GVL.Error_Code <= 3 THEN
        GVL.Error_Code := 0;
        Error_Code := 0;
    END_IF;
END_IF;

(* 2. HARD RESET INTERLOCK *)
IF Reset OR GVL.Reset THEN
    FOR i := 1 TO 6 DO
        Auto_Bin[i] := FALSE;
        auto_bin_cutoff[i] := FALSE;
        auto_bin_motor[i] := FALSE;
        Actual_Weights[i] := 0.0;
        GVL.Auto_Bin[i] := FALSE;
        GVL.auto_bin_cutoff[i] := FALSE;
        GVL.auto_bin_motor[i] := FALSE;
        GVL.Auto_Weights[i] := 0.0;
    END_FOR;
    
    (* Reset Recipe & Active Target Setpoints *)
    FOR i := 1 TO 20 DO
        GVL.Recipe_Weights[i] := 0.0;
    END_FOR;
    GVL.Auto_Total_Target_Weight := 0.0;
    GVL.Semi_Auto_Total_Target_Weight := 0.0;
    GVL.Auto_Material_Count := 0;
    GVL.Semi_Auto_Material_Count := 0;
    
    Sequence_Complete := FALSE;
    GVL.Auto_Sequence_Complete := FALSE;
    GVL.Semi_Auto_Sequence_Complete := FALSE;
    Active_Material_ID := 0;
    Active_Bin_ID := 0;
    Active_Target_Weight := 0.0;
    Active_Live_Weight := 0.0;
    GVL.Auto_Active_Target_Weight := 0.0;
    GVL.Auto_Active_Live_Weight := 0.0;
    Excess_Alarm := FALSE;
    Error_Code := 0;
    GVL.Error_Code := 0;
    GVL.Current_Batch_Cycle := 0;
    GVL.Completed_Batch_Cycles := 0;
    GVL.All_Cycles_Complete := FALSE;
    Auto_Completed_Batch_Cycles := 0;
    Auto_Current_Batch_Cycle := 0;
    Auto_All_Cycles_Complete := FALSE;
    GVL.Target_Batch_Cycles := 0;
    GVL.Start_Button := FALSE;
    GVL.Run := FALSE;
    GVL.Next_Cycle_Start := FALSE;
    Next_Cycle_Last := FALSE;
    Next_Cycle_Rising := FALSE;
    GVL.Auto_Active_Mat := 0;
    GVL.Auto_Active_Bin := 0;
    GVL.Auto_Excess_Alarm := FALSE;
    Current_Step := 0;
    Cycle_Manager_State := 0;
    Internal_FB_Start := FALSE;
    bin_last_weight := 0.0;
    Start_Sim_Weight := 0.0;
    Transition_Timer(IN := FALSE);
    Completion_Timer(IN := FALSE);
    Sim_Timer(IN := FALSE);
    Status_Message := 'Auto [Reset]: System Reset Complete - System Idle';
    RETURN;
END_IF;

(* 3. E-STOP PAUSE / HOLD LOGIC (NC Contact: FALSE = Pressed/Tripped, TRUE = Healthy) *)
IF NOT E_Stop_Active OR NOT GVL.E_Stop_Active THEN
    Paused_By_EStop := TRUE;
END_IF;

IF Paused_By_EStop THEN
    FOR i := 1 TO 6 DO
        Auto_Bin[i] := FALSE;
        auto_bin_cutoff[i] := FALSE;
        auto_bin_motor[i] := FALSE;
    END_FOR;
    IF NOT E_Stop_Active OR NOT GVL.E_Stop_Active THEN
        Status_Message := CONCAT('Auto [PAUSED]: E-Stop Active at Step ', INT_TO_STRING(Current_Step));
    ELSE
        Status_Message := CONCAT('Auto [HOLD]: E-Stop Cleared. Press Start to Resume Step ', INT_TO_STRING(Current_Step));
        IF Start_Button OR GVL.Start_Button THEN
            Paused_By_EStop := FALSE;
        END_IF;
    END_IF;
    Sim_Timer(IN := FALSE);
    Transition_Timer(IN := FALSE);
    Completion_Timer(IN := FALSE);
    RETURN;
END_IF;

(* 4. MASTER CYCLE MANAGER STATE MACHINE *)
CASE Cycle_Manager_State OF
    0: (* IDLE *)
        Internal_FB_Start := FALSE;
        GVL.Run := FALSE;
        GVL.Next_Cycle_Start := FALSE;
        GVL.Auto_Sequence_Complete := FALSE;
        
        IF GVL.Error_Code = 0 AND NOT (Start_Button OR GVL.Start_Button) THEN
            Status_Message := 'Auto [State 0 - Idle]: Ready - Waiting for Start Button';
        END_IF;
        
        IF Start_Button OR GVL.Start_Button THEN
            (* Use Target_Batch_Cycles from input, or fallback to GVL, or default to 1 *)
            IF Target_Batch_Cycles > 0 THEN
                GVL.Target_Batch_Cycles := Target_Batch_Cycles;
            ELSIF GVL.Target_Batch_Cycles <= 0 THEN
                GVL.Target_Batch_Cycles := 1;
            END_IF;
            
            IF NOT E_Stop_Active OR NOT GVL.E_Stop_Active THEN
                GVL.Run := FALSE;
                Status_Message := 'Auto [State 0]: Cannot Start - Emergency Stop Contact Open!';
            ELSIF (GVL.Auto_Initial_Tolerance > 0.0 AND (GVL.load_cell_auto > GVL.Auto_Initial_Tolerance OR GVL.load_cell_auto < (-GVL.Auto_Initial_Tolerance))) OR 
                  (GVL.Semi_Auto_Initial_Tolerance > 0.0 AND (GVL.load_cell_semi_auto > GVL.Semi_Auto_Initial_Tolerance OR GVL.load_cell_semi_auto < (-GVL.Semi_Auto_Initial_Tolerance))) THEN
                GVL.Run := FALSE;
                GVL.Error_Code := 4;
                Error_Code := 4;
                Status_Message := 'Auto [State 0]: Error 4 - Scale not zeroed (exceeds Initial Tolerance)!';
            ELSE
                GVL.Error_Code := 0;
                Error_Code := 0;
                GVL.Current_Batch_Cycle := 1;
                GVL.Completed_Batch_Cycles := 0;
                GVL.All_Cycles_Complete := FALSE;
                Auto_Completed_Batch_Cycles := 0;
                Auto_Current_Batch_Cycle := 1;
                Auto_All_Cycles_Complete := FALSE;
                GVL.Run := TRUE;
                Internal_FB_Start := TRUE;
                Cycle_Manager_State := 1;
                Current_Step := 0;
            END_IF;
        END_IF;
        
    1: (* RUNNING CYCLE *)
        Internal_FB_Start := TRUE;
        GVL.Run := TRUE;
        
        (* Interlock: While process is actively running, Next_Cycle_Start MUST be FALSE *)
        GVL.Next_Cycle_Start := FALSE;
        
        (* Both Auto and Semi-Auto must complete to finish the cycle *)
        IF Sequence_Complete AND GVL.Semi_Auto_Sequence_Complete THEN
            GVL.Completed_Batch_Cycles := GVL.Current_Batch_Cycle;
            Auto_Completed_Batch_Cycles := GVL.Current_Batch_Cycle;
            IF GVL.Current_Batch_Cycle < GVL.Target_Batch_Cycles AND GVL.Error_Code = 0 THEN
                Internal_FB_Start := FALSE;
                Cycle_Manager_State := 5; (* Go to pause/hold to wait for scale empty & Next_Cycle_Start *)
            ELSE
                Cycle_Manager_State := 4; (* All target cycles completed *)
            END_IF;
        END_IF;
        
    5: (* PAUSED BETWEEN CYCLES - WAITING FOR HOPPERS EMPTIED & NEXT CYCLE START *)
        Internal_FB_Start := FALSE;
        GVL.Run := TRUE;
        
        (* Determine effective empty weight threshold (defaults to 5.0 kg if <= 0.0) *)
        eff_empty_limit := Empty_Weight_Limit;
        IF eff_empty_limit <= 0.0 THEN
            eff_empty_limit := GVL.Empty_Weight_Limit;
        END_IF;
        IF eff_empty_limit <= 0.0 THEN
            eff_empty_limit := 5.0;
        END_IF;
        
        Status_Message := CONCAT('Auto [State 5]: Cycle ', CONCAT(INT_TO_STRING(GVL.Current_Batch_Cycle), ' Done. Empty scales < limit and trigger Next_Cycle_Start.'));
        
        (* Check ONLY on a new trigger pulse (rising edge) of Next_Cycle_Start *)
        IF Next_Cycle_Rising THEN
            (* Check both scales are below the empty weight limit at the moment of trigger *)
            IF (GVL.load_cell_auto < eff_empty_limit) AND (GVL.load_cell_semi_auto < eff_empty_limit) THEN
                (* Scale is empty: momentary reset of command, advance to next cycle *)
                GVL.Next_Cycle_Start := FALSE;
                Next_Cycle_Last := FALSE;
                GVL.Start_Button := TRUE; (* Keep Start_Button TRUE until all cycles are complete! *)
                GVL.Error_Code := 0;
                Error_Code := 0;
                GVL.Current_Batch_Cycle := GVL.Current_Batch_Cycle + 1;
                Auto_Current_Batch_Cycle := GVL.Current_Batch_Cycle;
                Sequence_Complete := FALSE;
                GVL.Auto_Sequence_Complete := FALSE;
                GVL.Semi_Auto_Sequence_Complete := FALSE;
                Current_Step := 0;
                Internal_FB_Start := TRUE;
                Cycle_Manager_State := 1;
                FOR i := 1 TO 6 DO
                    Actual_Weights[i] := 0.0;
                    Auto_Bin[i] := FALSE;
                    auto_bin_cutoff[i] := FALSE;
                    auto_bin_motor[i] := FALSE;
                END_FOR;
            ELSE
                (* Scale not empty yet: reject trigger, reset command, and wait for operator to trigger again *)
                GVL.Next_Cycle_Start := FALSE;
                Next_Cycle_Last := FALSE;
                Status_Message := CONCAT('Auto [State 5]: Scale weight exceeds limit (', CONCAT(REAL_TO_STRING(eff_empty_limit), ' kg)! Empty scales and trigger Next_Cycle_Start again.'));
            END_IF;
        END_IF;
        
    4: (* ALL CYCLES COMPLETE *)
        Internal_FB_Start := FALSE;
        GVL.Run := FALSE;
        GVL.Start_Button := FALSE;
        Auto_All_Cycles_Complete := TRUE;
        GVL.All_Cycles_Complete := TRUE;
        Sequence_Complete := TRUE;
        GVL.Auto_Sequence_Complete := TRUE;
        GVL.Semi_Auto_Sequence_Complete := TRUE;
        Status_Message := CONCAT('Auto [State 4 - Finished]: All ', CONCAT(INT_TO_STRING(GVL.Target_Batch_Cycles), ' Batch Cycles Completed Successfully'));
        IF Start_Button OR GVL.Start_Button THEN
            (* Reset flags for new batch start *)
            Current_Step := 0;
            Auto_All_Cycles_Complete := FALSE;
            GVL.All_Cycles_Complete := FALSE;
            Sequence_Complete := FALSE;
            GVL.Auto_Sequence_Complete := FALSE;
            GVL.Semi_Auto_Sequence_Complete := FALSE;
            Cycle_Manager_State := 0;
        END_IF;
END_CASE;

(* 5. AUTO SILOS 1..6 POURING SEQUENCE WITH DETAILED STATUS *)
IF Current_Step = 0 AND Internal_FB_Start THEN
    Current_Step := 1;
    bin_last_weight := load_cell_value;
    Sequence_Complete := FALSE;
    GVL.Auto_Sequence_Complete := FALSE;
    Excess_Alarm := FALSE;
    Error_Code := 0;
    FOR i := 1 TO 6 DO
        Actual_Weights[i] := 0.0;
        Auto_Bin[i] := FALSE;
        auto_bin_cutoff[i] := FALSE;
        auto_bin_motor[i] := FALSE;
    END_FOR;
END_IF;

CASE Current_Step OF
    0:
        Active_Material_ID := 0;
        Active_Bin_ID := 0;
        Excess_Alarm := FALSE;
        Sequence_Complete := FALSE;
        FOR i := 1 TO 6 DO
            Auto_Bin[i] := FALSE;
            auto_bin_cutoff[i] := FALSE;
            auto_bin_motor[i] := FALSE;
        END_FOR;
        Active_Target_Weight := GVL.Auto_Active_Target_Weight;
        Active_Live_Weight := 0.0;
        
    1..6:
        (* Skip any bin where Material Mapping is 0, > 20, or Recipe Weight is 0 *)
        WHILE Current_Step >= 1 AND Current_Step <= 6 DO
            Mat_Idx := Auto_Bin_Material_Mapping[Current_Step];
            IF Mat_Idx = 0 OR Mat_Idx > 20 OR GVL.Recipe_Weights[Mat_Idx] <= 0.0 THEN
                Auto_Bin[Current_Step] := FALSE;
                auto_bin_cutoff[Current_Step] := FALSE;
                auto_bin_motor[Current_Step] := FALSE;
                Actual_Weights[Current_Step] := 0.0;
                IF Current_Step = 6 THEN
                    Current_Step := 7;
                    EXIT;
                ELSE
                    Current_Step := Current_Step + 1;
                END_IF;
            ELSE
                EXIT; (* Valid active recipe silo found *)
            END_IF;
        END_WHILE;
        
        IF Current_Step = 7 THEN
            Active_Material_ID := 0;
            Active_Bin_ID := 0;
            Active_Target_Weight := 0.0;
            Active_Live_Weight := 0.0;
            GVL.Auto_Active_Target_Weight := 0.0;
            GVL.Auto_Active_Live_Weight := 0.0;
            Status_Message := 'Auto [Step 7]: Settling Delay in progress...';
            Completion_Timer(IN := TRUE, PT := Effective_Delay);
            IF Completion_Timer.Q THEN
                Completion_Timer(IN := FALSE);
                Current_Step := 8;
            END_IF;
        ELSE
            Mat_Idx := Auto_Bin_Material_Mapping[Current_Step];
            target_weight := GVL.Recipe_Weights[Mat_Idx];
            
            Active_Target_Weight := target_weight;
            GVL.Auto_Active_Target_Weight := target_weight;
            
            cutoff_trigger_weight := target_weight - Auto_Coarse_To_Fine_Speed[Current_Step];
            min_tol_weight := target_weight - Auto_Bin_Tolerance[Current_Step];
            max_tol_weight := target_weight + Auto_Bin_Tolerance[Current_Step];
            
            actual_bin := load_cell_value - bin_last_weight;
            IF actual_bin < 0.0 THEN
                actual_bin := 0.0;
            END_IF;
            Actual_Weights[Current_Step] := actual_bin;
            Active_Live_Weight := actual_bin;
            GVL.Auto_Active_Live_Weight := actual_bin;
            Active_Material_ID := Mat_Idx;
            Active_Bin_ID := Current_Step;
            
            IF load_cell_value > 500.0 THEN
                Error_Code := 21;
                GVL.Error_Code := 21;
                Status_Message := CONCAT('Auto [Step ', CONCAT(INT_TO_STRING(Current_Step), ']: STUCK - Error 21: Scale Overloaded (> 500 kg)!'));
                Sequence_Complete := TRUE;
                GVL.Auto_Sequence_Complete := TRUE;
                Paused_By_EStop := TRUE;
            END_IF;
            
            IF actual_bin < cutoff_trigger_weight THEN
                Auto_Bin[Current_Step] := TRUE;
                auto_bin_cutoff[Current_Step] := FALSE;
                auto_bin_motor[Current_Step] := TRUE;
                Excess_Alarm := FALSE;
                Status_Message := CONCAT('Auto [Step ', CONCAT(INT_TO_STRING(Current_Step), ']: Coarse Feeding'));
            ELSIF actual_bin < min_tol_weight THEN
                Auto_Bin[Current_Step] := FALSE;
                auto_bin_cutoff[Current_Step] := TRUE;
                auto_bin_motor[Current_Step] := TRUE;
                Excess_Alarm := FALSE;
                Status_Message := CONCAT('Auto [Step ', CONCAT(INT_TO_STRING(Current_Step), ']: Fine Feeding'));
            ELSIF actual_bin > max_tol_weight THEN
                Auto_Bin[Current_Step] := FALSE;
                auto_bin_cutoff[Current_Step] := FALSE;
                auto_bin_motor[Current_Step] := FALSE;
                IF Excess_Allowed THEN
                    Excess_Alarm := FALSE;
                    Status_Message := CONCAT('Auto [Step ', CONCAT(INT_TO_STRING(Current_Step), ']: Excess Allowed - Advancing'));
                    bin_last_weight := load_cell_value;
                    Active_Target_Weight := 0.0;
                    Active_Live_Weight := 0.0;
                    GVL.Auto_Active_Target_Weight := 0.0;
                    GVL.Auto_Active_Live_Weight := 0.0;
                    IF Current_Step = 6 THEN
                        Current_Step := 7;
                    ELSE
                        Current_Step := Current_Step + 1;
                    END_IF;
                ELSE
                    Excess_Alarm := TRUE;
                    Status_Message := CONCAT('Auto [Step ', CONCAT(INT_TO_STRING(Current_Step), ']: STUCK - Excess Weight! Reduce weight or enable Excess Allowed.'));
                END_IF;
            ELSE
                Auto_Bin[Current_Step] := FALSE;
                auto_bin_cutoff[Current_Step] := FALSE;
                auto_bin_motor[Current_Step] := FALSE;
                Excess_Alarm := FALSE;
                bin_last_weight := load_cell_value;
                Active_Target_Weight := 0.0;
                Active_Live_Weight := 0.0;
                GVL.Auto_Active_Target_Weight := 0.0;
                GVL.Auto_Active_Live_Weight := 0.0;
                Status_Message := CONCAT('Auto [Step ', CONCAT(INT_TO_STRING(Current_Step), ']: Target Reached - Advancing'));
                IF Current_Step = 6 THEN
                    Current_Step := 7;
                ELSE
                    Current_Step := Current_Step + 1;
                END_IF;
            END_IF;
        END_IF;

    7:
        Active_Material_ID := 0;
        Active_Bin_ID := 0;
        Excess_Alarm := FALSE;
        Status_Message := 'Auto [Step 7]: Settling Delay in progress...';
        Completion_Timer(IN := TRUE, PT := Effective_Delay);
        IF Completion_Timer.Q THEN
            Completion_Timer(IN := FALSE);
            Current_Step := 8;
        END_IF;
        
    8:
        Active_Material_ID := 0;
        Active_Bin_ID := 0;
        Excess_Alarm := FALSE;
        Sequence_Complete := TRUE;
        GVL.Auto_Sequence_Complete := TRUE;
        IF NOT GVL.Semi_Auto_Sequence_Complete THEN
            Status_Message := 'Auto [Step 8]: Auto Finished. Waiting for Semi-Auto to complete...';
        ELSE
            Status_Message := 'Auto [Step 8]: Cycle Sequences Complete';
        END_IF;
END_CASE;

(* Synchronize physical output arrays to GVL *)
FOR i := 1 TO 6 DO
    GVL.Auto_Bin[i] := Auto_Bin[i];
    GVL.auto_bin_cutoff[i] := auto_bin_cutoff[i];
    GVL.auto_bin_motor[i] := auto_bin_motor[i];
END_FOR;

(* Synchronize live cycle progress to outputs *)
Auto_Current_Batch_Cycle := GVL.Current_Batch_Cycle;
Auto_Completed_Batch_Cycles := GVL.Completed_Batch_Cycles;
Auto_All_Cycles_Complete := GVL.All_Cycles_Complete;

END_FUNCTION_BLOCK

